LIN {X 0,Y 181.229,Z 745.397,A -85,B 0,C 180,E1 -24524.153,E2 -24524.153} C_VEL
LIN {X 0,Y 171.019,Z 751.513,A -85,B 0,C 180,E1 -24527.303,E2 -24527.303} C_VEL
LIN {X 0,Y 164.032,Z 755.06,A -85,B 0,C 180,E1 -24530.003,E2 -24530.003} C_VEL
LIN {X 0,Y 155.67,Z 758.49,A -85,B 0,C 180,E1 -24534.057,E2 -24534.057} C_VEL
LIN {X 0,Y 149.094,Z 760.427,A -85,B 0,C 180,E1 -24538.049,E2 -24538.049} C_VEL
LIN {X 0,Y 142.632,Z 761.412,A -85,B 0,C 180,E1 -24543.67,E2 -24543.67} C_VEL
LIN {X 0,Y 138.275,Z 760.942,A -85,B 0,C 180,E1 -24549.154,E2 -24549.154} C_VEL
LIN {X 0,Y 135.73,Z 759.131,A -85,B 0,C 180,E1 -24554.99,E2 -24554.99} C_VEL
LIN {X 0,Y 134.847,Z 755.97,A -85,B 0,C 180,E1 -24561,E2 -24561} C_VEL
LIN {X 0,Y 135.175,Z 752.553,A -85,B 0,C 180,E1 -24565.522,E2 -24565.522} C_VEL
LIN {X 0,Y 135.672,Z 749.703,A -85,B 0,C 180,E1 -24568.511,E2 -24568.511} C_VEL
LIN {X 0,Y 135.626,Z 745.103,A -85,B 0,C 180,E1 -24572.222,E2 -24572.222} C_VEL
LIN {X 0,Y 135.586,Z 739.321,A -85,B 0,C 180,E1 -24575.945,E2 -24575.945} C_VEL
LIN {X 0,Y 135.696,Z 732.068,A -85,B 0,C 180,E1 -24579.732,E2 -24579.732} C_VEL
LIN {X 0,Y 136.328,Z 723.561,A -85,B 0,C 180,E1 -24583.409,E2 -24583.409} C_VEL
LIN {X 0,Y 136.604,Z 720.647,A -85,B 0,C 180,E1 -24584.52,E2 -24584.52} C_VEL
LIN {X 0,Y 137.564,Z 713.674,A -85,B 0,C 180,E1 -24589.39,E2 -24589.39} C_VEL
LIN {X 0,Y 139.573,Z 705.628,A -85,B 0,C 180,E1 -24593.75,E2 -24593.75} C_VEL
LIN {X 0,Y 141.934,Z 697.426,A -85,B 0,C 180,E1 -24597.254,E2 -24597.254} C_VEL
LIN {X 0,Y 144.902,Z 687.449,A -85,B 0,C 180,E1 -24600.609,E2 -24600.609} C_VEL
LIN {X 0,Y 148.196,Z 676.409,A -85,B 0,C 180,E1 -24603.451,E2 -24603.451} C_VEL
LIN {X 0,Y 150.997,Z 665.577,A -85,B 0,C 180,E1 -24605.571,E2 -24605.571} C_VEL
LIN {X 0,Y 153.57,Z 653.675,A -85,B 0,C 180,E1 -24607.322,E2 -24607.322} C_VEL
LIN {X 0,Y 155.586,Z 640.822,A -85,B 0,C 180,E1 -24608.701,E2 -24608.701} C_VEL
LIN {X 0,Y 156.825,Z 627.95,A -85,B 0,C 180,E1 -24609.612,E2 -24609.612} C_VEL
LIN {X 0,Y 157.546,Z 613.92,A -85,B 0,C 180,E1 -24610.242,E2 -24610.242} C_VEL
LIN {X 0,Y 155.056,Z 553.997,A -85,B 0,C 180,E1 -24614.23,E2 -24614.23} C_VEL
LIN {X 0,Y 151.174,Z 543.008,A -85,B 0,C 180,E1 -24616.002,E2 -24616.002} C_VEL
LIN {X 0,Y 146.403,Z 531.751,A -85,B 0,C 180,E1 -24618.235,E2 -24618.235} C_VEL
LIN {X 0,Y 142.973,Z 524.786,A -85,B 0,C 180,E1 -24619.906,E2 -24619.906} C_VEL
LIN {X 0,Y 140.588,Z 520.199,A -85,B 0,C 180,E1 -24621.118,E2 -24621.118} C_VEL
LIN {X 0,Y 138.476,Z 515.7,A -85,B 0,C 180,E1 -24622.479,E2 -24622.479} C_VEL
LIN {X 0,Y 136.204,Z 508.223,A -85,B 0,C 180,E1 -24628.068,E2 -24628.068} C_VEL
LIN {X 0,Y 136.07,Z 507.555,A -85,B 0,C 180,E1 -24628.901,E2 -24628.901} C_VEL
LIN {X 0,Y 136.136,Z 507.493,A -85,B 0,C 180,E1 -24632.313,E2 -24632.313} C_VEL
LIN {X 0,Y 136.233,Z 507.491,A -85,B 0,C 180,E1 -24638.83,E2 -24638.83} C_VEL
LIN {X 0,Y 136.273,Z 507.509,A -85,B 0,C 180,E1 -24645.055,E2 -24645.055} C_VEL
LIN {X 0,Y 136.486,Z 507.45,A -85,B 0,C 180,E1 -24648.113,E2 -24648.113} C_VEL
LIN {X 0,Y 136.58,Z 507.448,A -85,B 0,C 180,E1 -24651.119,E2 -24651.119} C_VEL
LIN {X 0,Y 137.122,Z 507.368,A -85,B 0,C 180,E1 -24659.999,E2 -24659.999} C_VEL
LIN {X 0,Y 136.566,Z 507.432,A -85,B 0,C 180,E1 -24668.88,E2 -24668.88} C_VEL
LIN {X 0,Y 136.479,Z 507.466,A -85,B 0,C 180,E1 -24671.954,E2 -24671.954} C_VEL
LIN {X 0,Y 136.239,Z 507.479,A -85,B 0,C 180,E1 -24678.029,E2 -24678.029} C_VEL
LIN {X 0,Y 136.186,Z 507.496,A -85,B 0,C 180,E1 -24681.75,E2 -24681.75} C_VEL
LIN {X 0,Y 136.088,Z 507.498,A -85,B 0,C 180,E1 -24688.618,E2 -24688.618} C_VEL
LIN {X 0,Y 136.059,Z 507.528,A -85,B 0,C 180,E1 -24694.623,E2 -24694.623} C_VEL
LIN {X 0,Y 136.025,Z 507.521,A -85,B 0,C 180,E1 -24699.203,E2 -24699.203} C_VEL
LIN {X 0,Y 136.035,Z 507.52,A -85,B 0,C 180,E1 -24703.681,E2 -24703.681} C_VEL
LIN {X 0,Y 136.08,Z 507.535,A -85,B 0,C 180,E1 -24707.832,E2 -24707.832} C_VEL
LIN {X 0,Y 136.125,Z 507.717,A -85,B 0,C 180,E1 -24711.986,E2 -24711.986} C_VEL
LIN {X 0,Y 136.369,Z 508.823,A -85,B 0,C 180,E1 -24712.654,E2 -24712.654} C_VEL
LIN {X 0,Y 137.916,Z 511.442,A -85,B 0,C 180,E1 -24713.555,E2 -24713.555} C_VEL
LIN {X 0,Y 139.347,Z 513.019,A -85,B 0,C 180,E1 -24714.26,E2 -24714.26} C_VEL
LIN {X 0,Y 141.795,Z 516.64,A -85,B 0,C 180,E1 -24715.486,E2 -24715.486} C_VEL
LIN {X 0,Y 147.533,Z 525.722,A -85,B 0,C 180,E1 -24718.149,E2 -24718.149} C_VEL
LIN {X 0,Y 153.564,Z 536.504,A -85,B 0,C 180,E1 -24720.727,E2 -24720.727} C_VEL
LIN {X 0,Y 159.744,Z 549.453,A -85,B 0,C 180,E1 -24723.189,E2 -24723.189} C_VEL
LIN {X 0,Y 160.42,Z 551.193,A -85,B 0,C 180,E1 -24723.46,E2 -24723.46} C_VEL
LIN {X 0,Y 158.812,Z 593.508,A -85,B 0,C 180,E1 -24725.453,E2 -24725.453} C_VEL
LIN {X 0,Y 157.758,Z 606.514,A -85,B 0,C 180,E1 -24726.542,E2 -24726.542} C_VEL
LIN {X 0,Y 156.131,Z 618.853,A -85,B 0,C 180,E1 -24728.032,E2 -24728.032} C_VEL
LIN {X 0,Y 153.973,Z 630.728,A -85,B 0,C 180,E1 -24729.986,E2 -24729.986} C_VEL
LIN {X 0,Y 151.336,Z 642.124,A -85,B 0,C 180,E1 -24732.436,E2 -24732.436} C_VEL
LIN {X 0,Y 148.657,Z 652.397,A -85,B 0,C 180,E1 -24735.284,E2 -24735.284} C_VEL
LIN {X 0,Y 146.153,Z 660.84,A -85,B 0,C 180,E1 -24738.212,E2 -24738.212} C_VEL
LIN {X 0,Y 143.314,Z 669.988,A -85,B 0,C 180,E1 -24742.254,E2 -24742.254} C_VEL
LIN {X 0,Y 140.794,Z 677.789,A -85,B 0,C 180,E1 -24746.676,E2 -24746.676} C_VEL
LIN {X 0,Y 138.812,Z 684.232,A -85,B 0,C 180,E1 -24751.455,E2 -24751.455} C_VEL
LIN {X 0,Y 137.647,Z 688.768,A -85,B 0,C 180,E1 -24755.866,E2 -24755.866} C_VEL
LIN {X 0,Y 137.075,Z 692.237,A -85,B 0,C 180,E1 -24760.343,E2 -24760.343} C_VEL
LIN {X 0,Y 137.153,Z 694.712,A -85,B 0,C 180,E1 -24764.85,E2 -24764.85} C_VEL
LIN {X 0,Y 138.239,Z 696.548,A -85,B 0,C 180,E1 -24770.852,E2 -24770.852} C_VEL
LIN {X 0,Y 139.867,Z 696.842,A -85,B 0,C 180,E1 -24775.252,E2 -24775.252} C_VEL
LIN {X 0,Y 142.219,Z 696.204,A -85,B 0,C 180,E1 -24779.62,E2 -24779.62} C_VEL
LIN {X 0,Y 144.114,Z 695.281,A -85,B 0,C 180,E1 -24782.447,E2 -24782.447} C_VEL
LIN {X 0,Y 146.406,Z 693.825,A -85,B 0,C 180,E1 -24785.31,E2 -24785.31} C_VEL
LIN {X 0,Y 150.148,Z 690.962,A -85,B 0,C 180,E1 -24789.196,E2 -24789.196} C_VEL
LIN {X 0,Y 155.29,Z 686.157,A -85,B 0,C 180,E1 -24793.606,E2 -24793.606} C_VEL
LIN {X 0,Y 157.794,Z 683.53,A -85,B 0,C 180,E1 -24795.454,E2 -24795.454} C_VEL
LIN {X 0,Y 149.569,Z 684.211,A -85,B 0,C 180,E1 -24798.866,E2 -24798.866} C_VEL
LIN {X 0,Y 140.091,Z 684.215,A -85,B 0,C 180,E1 -24804.767,E2 -24804.767} C_VEL
LIN {X 0,Y 139.135,Z 684.128,A -85,B 0,C 180,E1 -24805.92,E2 -24805.92} C_VEL
LIN {X 0,Y 138.913,Z 685.158,A -85,B 0,C 180,E1 -24806.512,E2 -24806.512} C_VEL
LIN {X 0,Y 137.09,Z 699.044,A -85,B 0,C 180,E1 -24810.341,E2 -24810.341} C_VEL
LIN {X 0,Y 135.806,Z 709.281,A -85,B 0,C 180,E1 -24813.905,E2 -24813.905} C_VEL
LIN {X 0,Y 134.865,Z 718.382,A -85,B 0,C 180,E1 -24817.803,E2 -24817.803} C_VEL
LIN {X 0,Y 134.137,Z 727.119,A -85,B 0,C 180,E1 -24822.467,E2 -24822.467} C_VEL
LIN {X 0,Y 133.895,Z 734.113,A -85,B 0,C 180,E1 -24827.111,E2 -24827.111} C_VEL
LIN {X 0,Y 134.285,Z 740.681,A -85,B 0,C 180,E1 -24832.608,E2 -24832.608} C_VEL
LIN {X 0,Y 135.926,Z 745.974,A -85,B 0,C 180,E1 -24838.52,E2 -24838.52} C_VEL
LIN {X 0,Y 138.001,Z 748.97,A -85,B 0,C 180,E1 -24842.92,E2 -24842.92} C_VEL
LIN {X 0,Y 142.183,Z 751.621,A -85,B 0,C 180,E1 -24848.529,E2 -24848.529} C_VEL
LIN {X 0,Y 147.77,Z 752.801,A -85,B 0,C 180,E1 -24853.758,E2 -24853.758} C_VEL
LIN {X 0,Y 154.776,Z 752.488,A -85,B 0,C 180,E1 -24858.534,E2 -24858.534} C_VEL
LIN {X 0,Y 162.866,Z 750.724,A -85,B 0,C 180,E1 -24862.854,E2 -24862.854} C_VEL
LIN {X 0,Y 172.025,Z 747.379,A -85,B 0,C 180,E1 -24866.706,E2 -24866.706} C_VEL
LIN {X 0,Y 179.516,Z 743.741,A -85,B 0,C 180,E1 -24869.3,E2 -24869.3} C_VEL
LIN {X 0,Y 187.457,Z 739.108,A -85,B 0,C 180,E1 -24871.661,E2 -24871.661} C_VEL
LIN {X 0,Y 196.841,Z 732.461,A -85,B 0,C 180,E1 -24874.06,E2 -24874.06} C_VEL
LIN {X 0,Y 205.986,Z 724.791,A -85,B 0,C 180,E1 -24876.055,E2 -24876.055} C_VEL
LIN {X 0,Y 211.642,Z 719.272,A -85,B 0,C 180,E1 -24877.154,E2 -24877.154} C_VEL
LIN {X 0,Y 212.865,Z 718.031,A -85,B 0,C 180,E1 -24877.586,E2 -24877.586} C_VEL
LIN {X 0,Y 203.705,Z 727.465,A -85,B 0,C 180,E1 -24879.075,E2 -24879.075} C_VEL
LIN {X 0,Y 199.807,Z 731.054,A -85,B 0,C 180,E1 -24879.811,E2 -24879.811} C_VEL
LIN {X 0,Y 195.562,Z 734.617,A -85,B 0,C 180,E1 -24880.454,E2 -24880.454} C_VEL
LIN {X 0,Y 187.687,Z 740.276,A -85,B 0,C 180,E1 -24881.137,E2 -24881.137} C_VEL
LIN {X 0,Y 179.639,Z 745.219,A -85,B 0,C 180,E1 -24881.969,E2 -24881.969} C_VEL
LIN {X 0,Y 175.187,Z 747.737,A -85,B 0,C 180,E1 -24882.866,E2 -24882.866} C_VEL
LIN {X 0,Y 165.932,Z 752.571,A -85,B 0,C 180,E1 -24885.66,E2 -24885.66} C_VEL
LIN {X 0,Y 158.69,Z 755.703,A -85,B 0,C 180,E1 -24888.365,E2 -24888.365} C_VEL
LIN {X 0,Y 149.985,Z 758.707,A -85,B 0,C 180,E1 -24892.466,E2 -24892.466} C_VEL
LIN {X 0,Y 142.55,Z 760.354,A -85,B 0,C 180,E1 -24896.946,E2 -24896.946} C_VEL
LIN {X 0,Y 136.305,Z 760.804,A -85,B 0,C 180,E1 -24902.346,E2 -24902.346} C_VEL
LIN {X 0,Y 131.704,Z 759.946,A -85,B 0,C 180,E1 -24908.061,E2 -24908.061} C_VEL
LIN {X 0,Y 128.973,Z 757.854,A -85,B 0,C 180,E1 -24914.184,E2 -24914.184} C_VEL
LIN {X 0,Y 128.004,Z 754.352,A -85,B 0,C 180,E1 -24920.514,E2 -24920.514} C_VEL
LIN {X 0,Y 128.351,Z 750.743,A -85,B 0,C 180,E1 -24925.284,E2 -24925.284} C_VEL
LIN {X 0,Y 128.845,Z 747.668,A -85,B 0,C 180,E1 -24928.432,E2 -24928.432} C_VEL
LIN {X 0,Y 128.784,Z 741.622,A -85,B 0,C 180,E1 -24933.123,E2 -24933.123} C_VEL
LIN {X 0,Y 128.752,Z 733.802,A -85,B 0,C 180,E1 -24937.838,E2 -24937.838} C_VEL
LIN {X 0,Y 129.123,Z 725.691,A -85,B 0,C 180,E1 -24941.783,E2 -24941.783} C_VEL
LIN {X 0,Y 129.477,Z 721.14,A -85,B 0,C 180,E1 -24943.732,E2 -24943.732} C_VEL
LIN {X 0,Y 130.27,Z 714.515,A -85,B 0,C 180,E1 -24948.881,E2 -24948.881} C_VEL
LIN {X 0,Y 132.17,Z 706.9,A -85,B 0,C 180,E1 -24953.498,E2 -24953.498} C_VEL
LIN {X 0,Y 134.642,Z 698.606,A -85,B 0,C 180,E1 -24957.454,E2 -24957.454} C_VEL
LIN {X 0,Y 137.731,Z 688.798,A -85,B 0,C 180,E1 -24961.102,E2 -24961.102} C_VEL
LIN {X 0,Y 141.14,Z 678.275,A -85,B 0,C 180,E1 -24964.063,E2 -24964.063} C_VEL
LIN {X 0,Y 144.364,Z 666.543,A -85,B 0,C 180,E1 -24966.604,E2 -24966.604} C_VEL
LIN {X 0,Y 147.032,Z 655.291,A -85,B 0,C 180,E1 -24968.411,E2 -24968.411} C_VEL
LIN {X 0,Y 149.255,Z 642.587,A -85,B 0,C 180,E1 -24969.902,E2 -24969.902} C_VEL
LIN {X 0,Y 150.774,Z 628.997,A -85,B 0,C 180,E1 -24970.988,E2 -24970.988} C_VEL
LIN {X 0,Y 151.631,Z 614.609,A -85,B 0,C 180,E1 -24971.675,E2 -24971.675} C_VEL
LIN {X 0,Y 149.494,Z 556.216,A -85,B 0,C 180,E1 -24975.709,E2 -24975.709} C_VEL
LIN {X 0,Y 145.779,Z 545.595,A -85,B 0,C 180,E1 -24977.549,E2 -24977.549} C_VEL
LIN {X 0,Y 140.792,Z 533.824,A -85,B 0,C 180,E1 -24980.095,E2 -24980.095} C_VEL
LIN {X 0,Y 136.234,Z 524.565,A -85,B 0,C 180,E1 -24982.57,E2 -24982.57} C_VEL
LIN {X 0,Y 133.372,Z 519.261,A -85,B 0,C 180,E1 -24984.224,E2 -24984.224} C_VEL
LIN {X 0,Y 130.784,Z 514.341,A -85,B 0,C 180,E1 -24985.998,E2 -24985.998} C_VEL
LIN {X 0,Y 129.054,Z 508.495,A -85,B 0,C 180,E1 -24990.93,E2 -24990.93} C_VEL
LIN {X 0,Y 129.02,Z 508.389,A -85,B 0,C 180,E1 -24994.164,E2 -24994.164} C_VEL
LIN {X 0,Y 129.097,Z 508.389,A -85,B 0,C 180,E1 -24997.725,E2 -24997.725} C_VEL
LIN {X 0,Y 129.149,Z 508.368,A -85,B 0,C 180,E1 -25000.942,E2 -25000.942} C_VEL
LIN {X 0,Y 129.405,Z 508.332,A -85,B 0,C 180,E1 -25007.818,E2 -25007.818} C_VEL
LIN {X 0,Y 129.505,Z 508.323,A -85,B 0,C 180,E1 -25010.629,E2 -25010.629} C_VEL
LIN {X 0,Y 130.077,Z 508.244,A -85,B 0,C 180,E1 -25019.999,E2 -25019.999} C_VEL
LIN {X 0,Y 129.495,Z 508.311,A -85,B 0,C 180,E1 -25029.369,E2 -25029.369} C_VEL
LIN {X 0,Y 129.381,Z 508.356,A -85,B 0,C 180,E1 -25032.548,E2 -25032.548} C_VEL
LIN {X 0,Y 129.147,Z 508.357,A -85,B 0,C 180,E1 -25039.056,E2 -25039.056} C_VEL
LIN {X 0,Y 129.096,Z 508.386,A -85,B 0,C 180,E1 -25042.399,E2 -25042.399} C_VEL
LIN {X 0,Y 129.018,Z 508.4,A -85,B 0,C 180,E1 -25045.834,E2 -25045.834} C_VEL
LIN {X 0,Y 129.004,Z 508.38,A -85,B 0,C 180,E1 -25049.36,E2 -25049.36} C_VEL
LIN {X 0,Y 128.969,Z 508.402,A -85,B 0,C 180,E1 -25055.184,E2 -25055.184} C_VEL
LIN {X 0,Y 128.97,Z 508.419,A -85,B 0,C 180,E1 -25060.836,E2 -25060.836} C_VEL
LIN {X 0,Y 129.011,Z 508.405,A -85,B 0,C 180,E1 -25067.09,E2 -25067.09} C_VEL
LIN {X 0,Y 129.064,Z 508.734,A -85,B 0,C 180,E1 -25068.766,E2 -25068.766} C_VEL
LIN {X 0,Y 129.373,Z 509.954,A -85,B 0,C 180,E1 -25069.421,E2 -25069.421} C_VEL
LIN {X 0,Y 131.114,Z 512.578,A -85,B 0,C 180,E1 -25070.551,E2 -25070.551} C_VEL
LIN {X 0,Y 132.475,Z 514.021,A -85,B 0,C 180,E1 -25071.327,E2 -25071.327} C_VEL
LIN {X 0,Y 134.708,Z 517.373,A -85,B 0,C 180,E1 -25072.622,E2 -25072.622} C_VEL
LIN {X 0,Y 136.153,Z 519.485,A -85,B 0,C 180,E1 -25073.412,E2 -25073.412} C_VEL
LIN {X 0,Y 141.454,Z 527.468,A -85,B 0,C 180,E1 -25076.104,E2 -25076.104} C_VEL
LIN {X 0,Y 148.043,Z 539.079,A -85,B 0,C 180,E1 -25079.168,E2 -25079.168} C_VEL
LIN {X 0,Y 154.555,Z 552.964,A -85,B 0,C 180,E1 -25081.98,E2 -25081.98} C_VEL
LIN {X 0,Y 152.942,Z 594.325,A -85,B 0,C 180,E1 -25084.01,E2 -25084.01} C_VEL
LIN {X 0,Y 151.835,Z 607.269,A -85,B 0,C 180,E1 -25085.122,E2 -25085.122} C_VEL
LIN {X 0,Y 150.051,Z 620.144,A -85,B 0,C 180,E1 -25086.727,E2 -25086.727} C_VEL
LIN {X 0,Y 147.77,Z 631.93,A -85,B 0,C 180,E1 -25088.742,E2 -25088.742} C_VEL
LIN {X 0,Y 144.996,Z 643.285,A -85,B 0,C 180,E1 -25091.275,E2 -25091.275} C_VEL
LIN {X 0,Y 142.163,Z 653.53,A -85,B 0,C 180,E1 -25094.228,E2 -25094.228} C_VEL
LIN {X 0,Y 139.26,Z 662.771,A -85,B 0,C 180,E1 -25097.62,E2 -25097.62} C_VEL
LIN {X 0,Y 136.318,Z 671.744,A -85,B 0,C 180,E1 -25101.854,E2 -25101.854} C_VEL
LIN {X 0,Y 133.809,Z 679.105,A -85,B 0,C 180,E1 -25106.295,E2 -25106.295} C_VEL
LIN {X 0,Y 132.201,Z 683.961,A -85,B 0,C 180,E1 -25110.005,E2 -25110.005} C_VEL
LIN {X 0,Y 130.85,Z 688.777,A -85,B 0,C 180,E1 -25114.626,E2 -25114.626} C_VEL
LIN {X 0,Y 130.116,Z 692.495,A -85,B 0,C 180,E1 -25119.33,E2 -25119.33} C_VEL
LIN {X 0,Y 130.036,Z 694.856,A -85,B 0,C 180,E1 -25123.389,E2 -25123.389} C_VEL
LIN {X 0,Y 130.668,Z 696.952,A -85,B 0,C 180,E1 -25128.832,E2 -25128.832} C_VEL
LIN {X 0,Y 131.492,Z 697.628,A -85,B 0,C 180,E1 -25131.976,E2 -25131.976} C_VEL
LIN {X 0,Y 133.16,Z 697.836,A -85,B 0,C 180,E1 -25136.206,E2 -25136.206} C_VEL
LIN {X 0,Y 135.932,Z 697.104,A -85,B 0,C 180,E1 -25141.138,E2 -25141.138} C_VEL
LIN {X 0,Y 138.017,Z 696.11,A -85,B 0,C 180,E1 -25144.071,E2 -25144.071} C_VEL
LIN {X 0,Y 140.431,Z 694.643,A -85,B 0,C 180,E1 -25146.915,E2 -25146.915} C_VEL
LIN {X 0,Y 144.56,Z 691.615,A -85,B 0,C 180,E1 -25151.026,E2 -25151.026} C_VEL
LIN {X 0,Y 149.604,Z 687.132,A -85,B 0,C 180,E1 -25155.199,E2 -25155.199} C_VEL
LIN {X 0,Y 144.92,Z 687.539,A -85,B 0,C 180,E1 -25157.241,E2 -25157.241} C_VEL
LIN {X 0,Y 136.909,Z 687.782,A -85,B 0,C 180,E1 -25161.977,E2 -25161.977} C_VEL
LIN {X 0,Y 131.712,Z 687.513,A -85,B 0,C 180,E1 -25166.387,E2 -25166.387} C_VEL
LIN {X 0,Y 131.451,Z 687.871,A -85,B 0,C 180,E1 -25167.113,E2 -25167.113} C_VEL
LIN {X 0,Y 131.075,Z 690.333,A -85,B 0,C 180,E1 -25167.932,E2 -25167.932} C_VEL
LIN {X 0,Y 129.543,Z 702.181,A -85,B 0,C 180,E1 -25171.661,E2 -25171.661} C_VEL
LIN {X 0,Y 128.315,Z 712.571,A -85,B 0,C 180,E1 -25175.747,E2 -25175.747} C_VEL
LIN {X 0,Y 127.444,Z 721.617,A -85,B 0,C 180,E1 -25180.152,E2 -25180.152} C_VEL
LIN {X 0,Y 126.996,Z 729.346,A -85,B 0,C 180,E1 -25184.761,E2 -25184.761} C_VEL
LIN {X 0,Y 126.92,Z 734.88,A -85,B 0,C 180,E1 -25188.826,E2 -25188.826} C_VEL
LIN {X 0,Y 127.469,Z 740.353,A -85,B 0,C 180,E1 -25193.67,E2 -25193.67} C_VEL
LIN {X 0,Y 128.753,Z 744.741,A -85,B 0,C 180,E1 -25198.437,E2 -25198.437} C_VEL
LIN {X 0,Y 130.814,Z 748.13,A -85,B 0,C 180,E1 -25203.081,E2 -25203.081} C_VEL
LIN {X 0,Y 135.324,Z 751.497,A -85,B 0,C 180,E1 -25209.307,E2 -25209.307} C_VEL
LIN {X 0,Y 140.756,Z 753.082,A -85,B 0,C 180,E1 -25214.458,E2 -25214.458} C_VEL
LIN {X 0,Y 147.945,Z 753.363,A -85,B 0,C 180,E1 -25219.423,E2 -25219.423} C_VEL
LIN {X 0,Y 156.26,Z 752.231,A -85,B 0,C 180,E1 -25223.879,E2 -25223.879} C_VEL
LIN {X 0,Y 165.706,Z 749.512,A -85,B 0,C 180,E1 -25227.811,E2 -25227.811} C_VEL
LIN {X 0,Y 173.368,Z 746.484,A -85,B 0,C 180,E1 -25230.447,E2 -25230.447} C_VEL
LIN {X 0,Y 181.509,Z 742.423,A -85,B 0,C 180,E1 -25232.826,E2 -25232.826} C_VEL
LIN {X 0,Y 190.977,Z 736.694,A -85,B 0,C 180,E1 -25235.189,E2 -25235.189} C_VEL
LIN {X 0,Y 199.017,Z 730.882,A -85,B 0,C 180,E1 -25236.895,E2 -25236.895} C_VEL
LIN {X 0,Y 199.44,Z 730.626,A -85,B 0,C 180,E1 -25237.541,E2 -25237.541} C_VEL
LIN {X 0,Y 189.089,Z 738.801,A -85,B 0,C 180,E1 -25239.531,E2 -25239.531} C_VEL
LIN {X 0,Y 179.189,Z 745.392,A -85,B 0,C 180,E1 -25241.819,E2 -25241.819} C_VEL
LIN {X 0,Y 175.187,Z 747.737,A -85,B 0,C 180,E1 -25242.866,E2 -25242.866} C_VEL
LIN {X 0,Y 170.662,Z 750.117,A -85,B 0,C 180,E1 -25243.871,E2 -25243.871} C_VEL
LIN {X 0,Y 162.216,Z 753.567,A -85,B 0,C 180,E1 -25245.23,E2 -25245.23} C_VEL
LIN {X 0,Y 153.855,Z 756.24,A -85,B 0,C 180,E1 -25246.84,E2 -25246.84} C_VEL
LIN {X 0,Y 149.549,Z 757.423,A -85,B 0,C 180,E1 -25248.257,E2 -25248.257} C_VEL
LIN {X 0,Y 140.228,Z 759.572,A -85,B 0,C 180,E1 -25253.023,E2 -25253.023} C_VEL
LIN {X 0,Y 133.109,Z 760.234,A -85,B 0,C 180,E1 -25258.125,E2 -25258.125} C_VEL
LIN {X 0,Y 127.483,Z 759.652,A -85,B 0,C 180,E1 -25263.825,E2 -25263.825} C_VEL
LIN {X 0,Y 123.531,Z 757.802,A -85,B 0,C 180,E1 -25270.035,E2 -25270.035} C_VEL
LIN {X 0,Y 121.49,Z 754.698,A -85,B 0,C 180,E1 -25276.615,E2 -25276.615} C_VEL
LIN {X 0,Y 121.362,Z 750.131,A -85,B 0,C 180,E1 -25283.344,E2 -25283.344} C_VEL
LIN {X 0,Y 122.042,Z 745.526,A -85,B 0,C 180,E1 -25288.345,E2 -25288.345} C_VEL
LIN {X 0,Y 121.949,Z 740.256,A -85,B 0,C 180,E1 -25292.472,E2 -25292.472} C_VEL
LIN {X 0,Y 121.881,Z 733.713,A -85,B 0,C 180,E1 -25296.617,E2 -25296.617} C_VEL
LIN {X 0,Y 122.225,Z 724.042,A -85,B 0,C 180,E1 -25301.572,E2 -25301.572} C_VEL
LIN {X 0,Y 122.352,Z 721.696,A -85,B 0,C 180,E1 -25302.658,E2 -25302.658} C_VEL
LIN {X 0,Y 123.016,Z 715.262,A -85,B 0,C 180,E1 -25308.308,E2 -25308.308} C_VEL
LIN {X 0,Y 124.753,Z 708.085,A -85,B 0,C 180,E1 -25313.219,E2 -25313.219} C_VEL
LIN {X 0,Y 127.58,Z 699.051,A -85,B 0,C 180,E1 -25317.959,E2 -25317.959} C_VEL
LIN {X 0,Y 130.947,Z 688.99,A -85,B 0,C 180,E1 -25321.999,E2 -25321.999} C_VEL
LIN {X 0,Y 134.448,Z 678.77,A -85,B 0,C 180,E1 -25325.093,E2 -25325.093} C_VEL
LIN {X 0,Y 137.798,Z 667.365,A -85,B 0,C 180,E1 -25327.729,E2 -25327.729} C_VEL
LIN {X 0,Y 140.772,Z 655.577,A -85,B 0,C 180,E1 -25329.76,E2 -25329.76} C_VEL
LIN {X 0,Y 143.235,Z 642.744,A -85,B 0,C 180,E1 -25331.358,E2 -25331.358} C_VEL
LIN {X 0,Y 144.873,Z 629.088,A -85,B 0,C 180,E1 -25332.517,E2 -25332.517} C_VEL
LIN {X 0,Y 145.807,Z 615.613,A -85,B 0,C 180,E1 -25333.193,E2 -25333.193} C_VEL
LIN {X 0,Y 144.01,Z 558.309,A -85,B 0,C 180,E1 -25337.319,E2 -25337.319} C_VEL
LIN {X 0,Y 139.806,Z 546.37,A -85,B 0,C 180,E1 -25339.594,E2 -25339.594} C_VEL
LIN {X 0,Y 134.923,Z 535.031,A -85,B 0,C 180,E1 -25342.349,E2 -25342.349} C_VEL
LIN {X 0,Y 129.935,Z 524.856,A -85,B 0,C 180,E1 -25345.405,E2 -25345.405} C_VEL
LIN {X 0,Y 126.142,Z 518.268,A -85,B 0,C 180,E1 -25347.923,E2 -25347.923} C_VEL
LIN {X 0,Y 123.07,Z 512.77,A -85,B 0,C 180,E1 -25350.375,E2 -25350.375} C_VEL
LIN {X 0,Y 122.019,Z 509.465,A -85,B 0,C 180,E1 -25353.487,E2 -25353.487} C_VEL
LIN {X 0,Y 122.038,Z 509.252,A -85,B 0,C 180,E1 -25359.784,E2 -25359.784} C_VEL
LIN {X 0,Y 122.253,Z 509.23,A -85,B 0,C 180,E1 -25366.705,E2 -25366.705} C_VEL
LIN {X 0,Y 122.435,Z 509.198,A -85,B 0,C 180,E1 -25370.083,E2 -25370.083} C_VEL
LIN {X 0,Y 122.592,Z 509.18,A -85,B 0,C 180,E1 -25376.712,E2 -25376.712} C_VEL
LIN {X 0,Y 123.031,Z 509.12,A -85,B 0,C 180,E1 -25379.999,E2 -25379.999} C_VEL
LIN {X 0,Y 122.399,Z 509.201,A -85,B 0,C 180,E1 -25387.145,E2 -25387.145} C_VEL
LIN {X 0,Y 122.35,Z 509.228,A -85,B 0,C 180,E1 -25392.471,E2 -25392.471} C_VEL
LIN {X 0,Y 122.105,Z 509.248,A -85,B 0,C 180,E1 -25396.724,E2 -25396.724} C_VEL
LIN {X 0,Y 122.016,Z 509.272,A -85,B 0,C 180,E1 -25402.857,E2 -25402.857} C_VEL
LIN {X 0,Y 121.93,Z 509.264,A -85,B 0,C 180,E1 -25407.458,E2 -25407.458} C_VEL
LIN {X 0,Y 121.895,Z 509.277,A -85,B 0,C 180,E1 -25411.258,E2 -25411.258} C_VEL
LIN {X 0,Y 121.887,Z 509.275,A -85,B 0,C 180,E1 -25416.183,E2 -25416.183} C_VEL
LIN {X 0,Y 121.902,Z 509.301,A -85,B 0,C 180,E1 -25421.463,E2 -25421.463} C_VEL
LIN {X 0,Y 121.945,Z 509.557,A -85,B 0,C 180,E1 -25424.645,E2 -25424.645} C_VEL
LIN {X 0,Y 122.237,Z 510.661,A -85,B 0,C 180,E1 -25425.409,E2 -25425.409} C_VEL
LIN {X 0,Y 123.774,Z 513.201,A -85,B 0,C 180,E1 -25426.633,E2 -25426.633} C_VEL
LIN {X 0,Y 125.622,Z 514.905,A -85,B 0,C 180,E1 -25427.868,E2 -25427.868} C_VEL
LIN {X 0,Y 127.726,Z 518.179,A -85,B 0,C 180,E1 -25429.313,E2 -25429.313} C_VEL
LIN {X 0,Y 129.124,Z 519.906,A -85,B 0,C 180,E1 -25430.181,E2 -25430.181} C_VEL
LIN {X 0,Y 134.391,Z 527.686,A -85,B 0,C 180,E1 -25433.269,E2 -25433.269} C_VEL
LIN {X 0,Y 139.727,Z 536.513,A -85,B 0,C 180,E1 -25436.079,E2 -25436.079} C_VEL
LIN {X 0,Y 144.984,Z 546.623,A -85,B 0,C 180,E1 -25438.634,E2 -25438.634} C_VEL
LIN {X 0,Y 148.918,Z 555.258,A -85,B 0,C 180,E1 -25440.452,E2 -25440.452} C_VEL
LIN {X 0,Y 147.152,Z 595.408,A -85,B 0,C 180,E1 -25442.472,E2 -25442.472} C_VEL
LIN {X 0,Y 145.981,Z 608.403,A -85,B 0,C 180,E1 -25443.632,E2 -25443.632} C_VEL
LIN {X 0,Y 144.229,Z 620.345,A -85,B 0,C 180,E1 -25445.153,E2 -25445.153} C_VEL
LIN {X 0,Y 141.992,Z 631.566,A -85,B 0,C 180,E1 -25447.065,E2 -25447.065} C_VEL
LIN {X 0,Y 139.058,Z 643.171,A -85,B 0,C 180,E1 -25449.673,E2 -25449.673} C_VEL
LIN {X 0,Y 136.047,Z 653.598,A -85,B 0,C 180,E1 -25452.726,E2 -25452.726} C_VEL
LIN {X 0,Y 132.961,Z 663.043,A -85,B 0,C 180,E1 -25456.245,E2 -25456.245} C_VEL
LIN {X 0,Y 129.789,Z 672.144,A -85,B 0,C 180,E1 -25460.656,E2 -25460.656} C_VEL
LIN {X 0,Y 127.306,Z 678.922,A -85,B 0,C 180,E1 -25464.826,E2 -25464.826} C_VEL
LIN {X 0,Y 125.094,Z 685.47,A -85,B 0,C 180,E1 -25470.005,E2 -25470.005} C_VEL
LIN {X 0,Y 123.705,Z 690.184,A -85,B 0,C 180,E1 -25474.894,E2 -25474.894} C_VEL
LIN {X 0,Y 123.041,Z 693.8,A -85,B 0,C 180,E1 -25479.872,E2 -25479.872} C_VEL
LIN {X 0,Y 123.006,Z 695.886,A -85,B 0,C 180,E1 -25483.766,E2 -25483.766} C_VEL
LIN {X 0,Y 123.855,Z 698.076,A -85,B 0,C 180,E1 -25489.911,E2 -25489.911} C_VEL
LIN {X 0,Y 124.8,Z 698.675,A -85,B 0,C 180,E1 -25493.222,E2 -25493.222} C_VEL
LIN {X 0,Y 127.77,Z 698.621,A -85,B 0,C 180,E1 -25499.678,E2 -25499.678} C_VEL
LIN {X 0,Y 129.77,Z 697.996,A -85,B 0,C 180,E1 -25502.797,E2 -25502.797} C_VEL
LIN {X 0,Y 134.093,Z 695.755,A -85,B 0,C 180,E1 -25508.173,E2 -25508.173} C_VEL
LIN {X 0,Y 139.123,Z 692.27,A -85,B 0,C 180,E1 -25513.004,E2 -25513.004} C_VEL
LIN {X 0,Y 140.752,Z 690.983,A -85,B 0,C 180,E1 -25514.356,E2 -25514.356} C_VEL
LIN {X 0,Y 140.256,Z 690.513,A -85,B 0,C 180,E1 -25515.453,E2 -25515.453} C_VEL
LIN {X 0,Y 131.964,Z 690.972,A -85,B 0,C 180,E1 -25520.278,E2 -25520.278} C_VEL
LIN {X 0,Y 124,Z 690.732,A -85,B 0,C 180,E1 -25527.594,E2 -25527.594} C_VEL
LIN {X 0,Y 123.794,Z 691.458,A -85,B 0,C 180,E1 -25528.393,E2 -25528.393} C_VEL
LIN {X 0,Y 122.116,Z 704.804,A -85,B 0,C 180,E1 -25533.051,E2 -25533.051} C_VEL
LIN {X 0,Y 120.926,Z 715.427,A -85,B 0,C 180,E1 -25537.703,E2 -25537.703} C_VEL
LIN {X 0,Y 120.25,Z 723.579,A -85,B 0,C 180,E1 -25542.133,E2 -25542.133} C_VEL
LIN {X 0,Y 119.96,Z 731.262,A -85,B 0,C 180,E1 -25547.31,E2 -25547.31} C_VEL
LIN {X 0,Y 120.35,Z 738.394,A -85,B 0,C 180,E1 -25553.294,E2 -25553.294} C_VEL
LIN {X 0,Y 121.613,Z 743.231,A -85,B 0,C 180,E1 -25558.345,E2 -25558.345} C_VEL
LIN {X 0,Y 124.543,Z 748.152,A -85,B 0,C 180,E1 -25564.857,E2 -25564.857} C_VEL
LIN {X 0,Y 128.568,Z 751.203,A -85,B 0,C 180,E1 -25570.253,E2 -25570.253} C_VEL
LIN {X 0,Y 133.747,Z 753.126,A -85,B 0,C 180,E1 -25575.234,E2 -25575.234} C_VEL
LIN {X 0,Y 141.132,Z 754.006,A -85,B 0,C 180,E1 -25580.402,E2 -25580.402} C_VEL
LIN {X 0,Y 149.677,Z 753.484,A -85,B 0,C 180,E1 -25584.999,E2 -25584.999} C_VEL
LIN {X 0,Y 159.409,Z 751.436,A -85,B 0,C 180,E1 -25589.011,E2 -25589.011} C_VEL
LIN {X 0,Y 167.255,Z 748.929,A -85,B 0,C 180,E1 -25591.686,E2 -25591.686} C_VEL
LIN {X 0,Y 178.797,Z 743.963,A -85,B 0,C 180,E1 -25594.885,E2 -25594.885} C_VEL
LIN {X 0,Y 187.367,Z 739.251,A -85,B 0,C 180,E1 -25596.881,E2 -25596.881} C_VEL
LIN {X 0,Y 186.244,Z 740.052,A -85,B 0,C 180,E1 -25597.58,E2 -25597.58} C_VEL
LIN {X 0,Y 176.718,Z 745.884,A -85,B 0,C 180,E1 -25599.607,E2 -25599.607} C_VEL
LIN {X 0,Y 166.294,Z 751.171,A -85,B 0,C 180,E1 -25602.298,E2 -25602.298} C_VEL
LIN {X 0,Y 158.435,Z 754.477,A -85,B 0,C 180,E1 -25604.781,E2 -25604.781} C_VEL
LIN {X 0,Y 149.549,Z 757.423,A -85,B 0,C 180,E1 -25608.257,E2 -25608.257} C_VEL
LIN {X 0,Y 145.321,Z 758.452,A -85,B 0,C 180,E1 -25609.814,E2 -25609.814} C_VEL
LIN {X 0,Y 137.369,Z 759.459,A -85,B 0,C 180,E1 -25612.181,E2 -25612.181} C_VEL
LIN {X 0,Y 129.861,Z 759.676,A -85,B 0,C 180,E1 -25614.917,E2 -25614.917} C_VEL
LIN {X 0,Y 126.438,Z 759.483,A -85,B 0,C 180,E1 -25617.047,E2 -25617.047} C_VEL
LIN {X 0,Y 121.19,Z 758.61,A -85,B 0,C 180,E1 -25622.353,E2 -25622.353} C_VEL
LIN {X 0,Y 116.988,Z 756.454,A -85,B 0,C 180,E1 -25628.866,E2 -25628.866} C_VEL
LIN {X 0,Y 114.79,Z 752.958,A -85,B 0,C 180,E1 -25635.818,E2 -25635.818} C_VEL
LIN {X 0,Y 114.636,Z 748.069,A -85,B 0,C 180,E1 -25642.951,E2 -25642.951} C_VEL
LIN {X 0,Y 115.112,Z 744.959,A -85,B 0,C 180,E1 -25646.494,E2 -25646.494} C_VEL
LIN {X 0,Y 115.254,Z 742.131,A -85,B 0,C 180,E1 -25649.121,E2 -25649.121} C_VEL
LIN {X 0,Y 115.073,Z 736.306,A -85,B 0,C 180,E1 -25653.496,E2 -25653.496} C_VEL
LIN {X 0,Y 114.991,Z 729.05,A -85,B 0,C 180,E1 -25657.898,E2 -25657.898} C_VEL
LIN {X 0,Y 115.326,Z 722.07,A -85,B 0,C 180,E1 -25661.543,E2 -25661.543} C_VEL
LIN {X 0,Y 115.739,Z 715.909,A -85,B 0,C 180,E1 -25667.669,E2 -25667.669} C_VEL
LIN {X 0,Y 117.376,Z 709.083,A -85,B 0,C 180,E1 -25672.898,E2 -25672.898} C_VEL
LIN {X 0,Y 120.134,Z 700.658,A -85,B 0,C 180,E1 -25677.899,E2 -25677.899} C_VEL
LIN {X 0,Y 123.175,Z 692.07,A -85,B 0,C 180,E1 -25681.849,E2 -25681.849} C_VEL
LIN {X 0,Y 126.957,Z 681.533,A -85,B 0,C 180,E1 -25685.532,E2 -25685.532} C_VEL
LIN {X 0,Y 130.838,Z 669.662,A -85,B 0,C 180,E1 -25688.634,E2 -25688.634} C_VEL
LIN {X 0,Y 134.102,Z 657.803,A -85,B 0,C 180,E1 -25690.92,E2 -25690.92} C_VEL
LIN {X 0,Y 136.691,Z 645.977,A -85,B 0,C 180,E1 -25692.583,E2 -25692.583} C_VEL
LIN {X 0,Y 138.701,Z 632.742,A -85,B 0,C 180,E1 -25693.907,E2 -25693.907} C_VEL
LIN {X 0,Y 139.93,Z 619.903,A -85,B 0,C 180,E1 -25694.673,E2 -25694.673} C_VEL
LIN {X 0,Y 139.963,Z 611.462,A -85,B 0,C 180,E1 -25695.205,E2 -25695.205} C_VEL
LIN {X 0,Y 138.615,Z 560.34,A -85,B 0,C 180,E1 -25699.072,E2 -25699.072} C_VEL
LIN {X 0,Y 134.319,Z 548.06,A -85,B 0,C 180,E1 -25701.629,E2 -25701.629} C_VEL
LIN {X 0,Y 129.756,Z 537.481,A -85,B 0,C 180,E1 -25704.476,E2 -25704.476} C_VEL
LIN {X 0,Y 125.553,Z 528.831,A -85,B 0,C 180,E1 -25707.324,E2 -25707.324} C_VEL
LIN {X 0,Y 122.489,Z 523.211,A -85,B 0,C 180,E1 -25709.576,E2 -25709.576} C_VEL
LIN {X 0,Y 118.998,Z 517.241,A -85,B 0,C 180,E1 -25712.399,E2 -25712.399} C_VEL
LIN {X 0,Y 115.282,Z 511.674,A -85,B 0,C 180,E1 -25715.847,E2 -25715.847} C_VEL
LIN {X 0,Y 115.001,Z 510.433,A -85,B 0,C 180,E1 -25716.885,E2 -25716.885} C_VEL
LIN {X 0,Y 114.971,Z 510.138,A -85,B 0,C 180,E1 -25718.482,E2 -25718.482} C_VEL
LIN {X 0,Y 115.137,Z 510.125,A -85,B 0,C 180,E1 -25725.866,E2 -25725.866} C_VEL
LIN {X 0,Y 115.353,Z 510.077,A -85,B 0,C 180,E1 -25729.467,E2 -25729.467} C_VEL
LIN {X 0,Y 115.518,Z 510.061,A -85,B 0,C 180,E1 -25736.511,E2 -25736.511} C_VEL
LIN {X 0,Y 115.983,Z 509.996,A -85,B 0,C 180,E1 -25739.999,E2 -25739.999} C_VEL
LIN {X 0,Y 115.367,Z 510.076,A -85,B 0,C 180,E1 -25747.035,E2 -25747.035} C_VEL
LIN {X 0,Y 115.271,Z 510.111,A -85,B 0,C 180,E1 -25752.735,E2 -25752.735} C_VEL
LIN {X 0,Y 115.005,Z 510.121,A -85,B 0,C 180,E1 -25757.79,E2 -25757.79} C_VEL
LIN {X 0,Y 114.936,Z 510.162,A -85,B 0,C 180,E1 -25763.495,E2 -25763.495} C_VEL
LIN {X 0,Y 114.85,Z 510.151,A -85,B 0,C 180,E1 -25771.064,E2 -25771.064} C_VEL
LIN {X 0,Y 114.827,Z 510.239,A -85,B 0,C 180,E1 -25778.853,E2 -25778.853} C_VEL
LIN {X 0,Y 115.001,Z 511.064,A -85,B 0,C 180,E1 -25780.201,E2 -25780.201} C_VEL
LIN {X 0,Y 116.564,Z 513.994,A -85,B 0,C 180,E1 -25781.896,E2 -25781.896} C_VEL
LIN {X 0,Y 118.91,Z 515.962,A -85,B 0,C 180,E1 -25783.797,E2 -25783.797} C_VEL
LIN {X 0,Y 120.856,Z 519.153,A -85,B 0,C 180,E1 -25785.421,E2 -25785.421} C_VEL
LIN {X 0,Y 122.572,Z 521.004,A -85,B 0,C 180,E1 -25786.668,E2 -25786.668} C_VEL
LIN {X 0,Y 125.037,Z 524.484,A -85,B 0,C 180,E1 -25788.415,E2 -25788.415} C_VEL
LIN {X 0,Y 130.672,Z 533.023,A -85,B 0,C 180,E1 -25792.006,E2 -25792.006} C_VEL
LIN {X 0,Y 135.568,Z 541.402,A -85,B 0,C 180,E1 -25794.789,E2 -25794.789} C_VEL
LIN {X 0,Y 140.481,Z 551.149,A -85,B 0,C 180,E1 -25797.364,E2 -25797.364} C_VEL
LIN {X 0,Y 143.299,Z 557.454,A -85,B 0,C 180,E1 -25798.767,E2 -25798.767} C_VEL
LIN {X 0,Y 141.432,Z 596.902,A -85,B 0,C 180,E1 -25800.835,E2 -25800.835} C_VEL
LIN {X 0,Y 140.059,Z 610.651,A -85,B 0,C 180,E1 -25802.13,E2 -25802.13} C_VEL
LIN {X 0,Y 138.13,Z 622.704,A -85,B 0,C 180,E1 -25803.773,E2 -25803.773} C_VEL
LIN {X 0,Y 135.561,Z 634.352,A -85,B 0,C 180,E1 -25805.91,E2 -25805.91} C_VEL
LIN {X 0,Y 132.493,Z 645.618,A -85,B 0,C 180,E1 -25808.618,E2 -25808.618} C_VEL
LIN {X 0,Y 129.329,Z 655.791,A -85,B 0,C 180,E1 -25811.798,E2 -25811.798} C_VEL
LIN {X 0,Y 126.104,Z 664.965,A -85,B 0,C 180,E1 -25815.481,E2 -25815.481} C_VEL
LIN {X 0,Y 122.795,Z 673.908,A -85,B 0,C 180,E1 -25820.119,E2 -25820.119} C_VEL
LIN {X 0,Y 119.872,Z 681.604,A -85,B 0,C 180,E1 -25825.324,E2 -25825.324} C_VEL
LIN {X 0,Y 117.963,Z 686.951,A -85,B 0,C 180,E1 -25830.006,E2 -25830.006} C_VEL
LIN {X 0,Y 116.551,Z 691.554,A -85,B 0,C 180,E1 -25835.195,E2 -25835.195} C_VEL
LIN {X 0,Y 115.952,Z 695.073,A -85,B 0,C 180,E1 -25840.482,E2 -25840.482} C_VEL
LIN {X 0,Y 115.996,Z 696.925,A -85,B 0,C 180,E1 -25844.212,E2 -25844.212} C_VEL
LIN {X 0,Y 117.081,Z 699.188,A -85,B 0,C 180,E1 -25851.116,E2 -25851.116} C_VEL
LIN {X 0,Y 119.665,Z 699.833,A -85,B 0,C 180,E1 -25858.03,E2 -25858.03} C_VEL
LIN {X 0,Y 121.513,Z 699.564,A -85,B 0,C 180,E1 -25861.374,E2 -25861.374} C_VEL
LIN {X 0,Y 123.719,Z 698.857,A -85,B 0,C 180,E1 -25864.622,E2 -25864.622} C_VEL
LIN {X 0,Y 128.08,Z 696.728,A -85,B 0,C 180,E1 -25869.809,E2 -25869.809} C_VEL
LIN {X 0,Y 132.207,Z 694.14,A -85,B 0,C 180,E1 -25873.721,E2 -25873.721} C_VEL
LIN {X 0,Y 132.448,Z 693.411,A -85,B 0,C 180,E1 -25875.122,E2 -25875.122} C_VEL
LIN {X 0,Y 123.324,Z 693.937,A -85,B 0,C 180,E1 -25881.182,E2 -25881.182} C_VEL
LIN {X 0,Y 116.455,Z 693.802,A -85,B 0,C 180,E1 -25888.635,E2 -25888.635} C_VEL
LIN {X 0,Y 116.25,Z 694.18,A -85,B 0,C 180,E1 -25889.457,E2 -25889.457} C_VEL
LIN {X 0,Y 114.644,Z 707.164,A -85,B 0,C 180,E1 -25894.59,E2 -25894.59} C_VEL
LIN {X 0,Y 113.732,Z 716.643,A -85,B 0,C 180,E1 -25899.189,E2 -25899.189} C_VEL
LIN {X 0,Y 113.143,Z 725.749,A -85,B 0,C 180,E1 -25904.694,E2 -25904.694} C_VEL
LIN {X 0,Y 113.093,Z 733.073,A -85,B 0,C 180,E1 -25910.162,E2 -25910.162} C_VEL
LIN {X 0,Y 114.014,Z 739.817,A -85,B 0,C 180,E1 -25916.467,E2 -25916.467} C_VEL
LIN {X 0,Y 116.49,Z 745.734,A -85,B 0,C 180,E1 -25923.46,E2 -25923.46} C_VEL
LIN {X 0,Y 120.805,Z 750.076,A -85,B 0,C 180,E1 -25930.053,E2 -25930.053} C_VEL
LIN {X 0,Y 126.781,Z 752.935,A -85,B 0,C 180,E1 -25936.093,E2 -25936.093} C_VEL
LIN {X 0,Y 134.354,Z 754.401,A -85,B 0,C 180,E1 -25941.481,E2 -25941.481} C_VEL
LIN {X 0,Y 143.144,Z 754.486,A -85,B 0,C 180,E1 -25946.225,E2 -25946.225} C_VEL
LIN {X 0,Y 153.149,Z 753.089,A -85,B 0,C 180,E1 -25950.318,E2 -25950.318} C_VEL
LIN {X 0,Y 158.417,Z 751.859,A -85,B 0,C 180,E1 -25952.167,E2 -25952.167} C_VEL
LIN {X 0,Y 169.763,Z 748.238,A -85,B 0,C 180,E1 -25955.422,E2 -25955.422} C_VEL
LIN {X 0,Y 176.058,Z 745.585,A -85,B 0,C 180,E1 -25957.019,E2 -25957.019} C_VEL
LIN {X 0,Y 164.452,Z 751.12,A -85,B 0,C 180,E1 -25959.708,E2 -25959.708} C_VEL
LIN {X 0,Y 153.536,Z 755.133,A -85,B 0,C 180,E1 -25962.907,E2 -25962.907} C_VEL
LIN {X 0,Y 143.556,Z 757.835,A -85,B 0,C 180,E1 -25966.728,E2 -25966.728} C_VEL
LIN {X 0,Y 134.626,Z 759.292,A -85,B 0,C 180,E1 -25971.206,E2 -25971.206} C_VEL
LIN {X 0,Y 127.153,Z 759.552,A -85,B 0,C 180,E1 -25976.44,E2 -25976.44} C_VEL
LIN {X 0,Y 126.438,Z 759.483,A -85,B 0,C 180,E1 -25977.047,E2 -25977.047} C_VEL
LIN {X 0,Y 123.262,Z 759.133,A -85,B 0,C 180,E1 -25979.319,E2 -25979.319} C_VEL
LIN {X 0,Y 117.061,Z 757.641,A -85,B 0,C 180,E1 -25982.931,E2 -25982.931} C_VEL
LIN {X 0,Y 111.569,Z 755.406,A -85,B 0,C 180,E1 -25986.913,E2 -25986.913} C_VEL
LIN {X 0,Y 109.617,Z 753.896,A -85,B 0,C 180,E1 -25989.702,E2 -25989.702} C_VEL
LIN {X 0,Y 108.151,Z 751.114,A -85,B 0,C 180,E1 -25994.928,E2 -25994.928} C_VEL
LIN {X 0,Y 107.943,Z 745.874,A -85,B 0,C 180,E1 -26002.512,E2 -26002.512} C_VEL
LIN {X 0,Y 108.446,Z 742.576,A -85,B 0,C 180,E1 -26006.278,E2 -26006.278} C_VEL
LIN {X 0,Y 108.484,Z 738.416,A -85,B 0,C 180,E1 -26009.994,E2 -26009.994} C_VEL
LIN {X 0,Y 108.246,Z 731.884,A -85,B 0,C 180,E1 -26014.649,E2 -26014.649} C_VEL
LIN {X 0,Y 108.356,Z 722.327,A -85,B 0,C 180,E1 -26020.268,E2 -26020.268} C_VEL
LIN {X 0,Y 108.527,Z 716.427,A -85,B 0,C 180,E1 -26026.936,E2 -26026.936} C_VEL
LIN {X 0,Y 110.046,Z 710.007,A -85,B 0,C 180,E1 -26032.524,E2 -26032.524} C_VEL
LIN {X 0,Y 112.683,Z 702.044,A -85,B 0,C 180,E1 -26037.883,E2 -26037.883} C_VEL
LIN {X 0,Y 115.668,Z 694.065,A -85,B 0,C 180,E1 -26042.027,E2 -26042.027} C_VEL
LIN {X 0,Y 119.477,Z 684.041,A -85,B 0,C 180,E1 -26046.024,E2 -26046.024} C_VEL
LIN {X 0,Y 123.434,Z 673.117,A -85,B 0,C 180,E1 -26049.296,E2 -26049.296} C_VEL
LIN {X 0,Y 126.775,Z 662.471,A -85,B 0,C 180,E1 -26051.693,E2 -26051.693} C_VEL
LIN {X 0,Y 130.062,Z 649.63,A -85,B 0,C 180,E1 -26053.807,E2 -26053.807} C_VEL
LIN {X 0,Y 132.485,Z 636.647,A -85,B 0,C 180,E1 -26055.334,E2 -26055.334} C_VEL
LIN {X 0,Y 134.044,Z 623.561,A -85,B 0,C 180,E1 -26056.315,E2 -26056.315} C_VEL
LIN {X 0,Y 134.48,Z 614.683,A -85,B 0,C 180,E1 -26056.82,E2 -26056.82} C_VEL
LIN {X 0,Y 133.429,Z 562.638,A -85,B 0,C 180,E1 -26060.917,E2 -26060.917} C_VEL
LIN {X 0,Y 129.163,Z 550.337,A -85,B 0,C 180,E1 -26063.719,E2 -26063.719} C_VEL
LIN {X 0,Y 124.697,Z 539.651,A -85,B 0,C 180,E1 -26066.846,E2 -26066.846} C_VEL
LIN {X 0,Y 121.402,Z 532.879,A -85,B 0,C 180,E1 -26069.324,E2 -26069.324} C_VEL
LIN {X 0,Y 118.846,Z 528.047,A -85,B 0,C 180,E1 -26071.403,E2 -26071.403} C_VEL
LIN {X 0,Y 115.883,Z 522.697,A -85,B 0,C 180,E1 -26074.035,E2 -26074.035} C_VEL
LIN {X 0,Y 112.225,Z 516.964,A -85,B 0,C 180,E1 -26077.668,E2 -26077.668} C_VEL
LIN {X 0,Y 109.151,Z 514.236,A -85,B 0,C 180,E1 -26080.975,E2 -26080.975} C_VEL
LIN {X 0,Y 108.046,Z 511.582,A -85,B 0,C 180,E1 -26082.978,E2 -26082.978} C_VEL
LIN {X 0,Y 107.994,Z 511.057,A -85,B 0,C 180,E1 -26084.427,E2 -26084.427} C_VEL
LIN {X 0,Y 108.277,Z 510.957,A -85,B 0,C 180,E1 -26088.77,E2 -26088.77} C_VEL
LIN {X 0,Y 108.443,Z 510.942,A -85,B 0,C 180,E1 -26096.283,E2 -26096.283} C_VEL
LIN {X 0,Y 108.909,Z 510.876,A -85,B 0,C 180,E1 -26099.999,E2 -26099.999} C_VEL
LIN {X 0,Y 108.31,Z 510.95,A -85,B 0,C 180,E1 -26107.455,E2 -26107.455} C_VEL
LIN {X 0,Y 108.185,Z 510.995,A -85,B 0,C 180,E1 -26113.013,E2 -26113.013} C_VEL
LIN {X 0,Y 107.896,Z 511,A -85,B 0,C 180,E1 -26119.006,E2 -26119.006} C_VEL
LIN {X 0,Y 107.846,Z 511.051,A -85,B 0,C 180,E1 -26124.186,E2 -26124.186} C_VEL
LIN {X 0,Y 107.796,Z 511.229,A -85,B 0,C 180,E1 -26132.481,E2 -26132.481} C_VEL
LIN {X 0,Y 107.972,Z 512.113,A -85,B 0,C 180,E1 -26133.726,E2 -26133.726} C_VEL
LIN {X 0,Y 109.291,Z 514.703,A -85,B 0,C 180,E1 -26135.634,E2 -26135.634} C_VEL
LIN {X 0,Y 112.245,Z 517.118,A -85,B 0,C 180,E1 -26138.764,E2 -26138.764} C_VEL
LIN {X 0,Y 114.233,Z 520.339,A -85,B 0,C 180,E1 -26140.818,E2 -26140.818} C_VEL
LIN {X 0,Y 116.127,Z 522.204,A -85,B 0,C 180,E1 -26142.489,E2 -26142.489} C_VEL
LIN {X 0,Y 118.651,Z 525.772,A -85,B 0,C 180,E1 -26144.649,E2 -26144.649} C_VEL
LIN {X 0,Y 123.013,Z 532.06,A -85,B 0,C 180,E1 -26147.962,E2 -26147.962} C_VEL
LIN {X 0,Y 127.952,Z 539.913,A -85,B 0,C 180,E1 -26151.263,E2 -26151.263} C_VEL
LIN {X 0,Y 133.092,Z 549.393,A -85,B 0,C 180,E1 -26154.351,E2 -26154.351} C_VEL
LIN {X 0,Y 137.797,Z 559.649,A -85,B 0,C 180,E1 -26156.963,E2 -26156.963} C_VEL
LIN {X 0,Y 135.899,Z 597.54,A -85,B 0,C 180,E1 -26159.01,E2 -26159.01} C_VEL
LIN {X 0,Y 134.47,Z 611.18,A -85,B 0,C 180,E1 -26160.318,E2 -26160.318} C_VEL
LIN {X 0,Y 132.29,Z 623.927,A -85,B 0,C 180,E1 -26162.091,E2 -26162.091} C_VEL
LIN {X 0,Y 129.615,Z 635.513,A -85,B 0,C 180,E1 -26164.299,E2 -26164.299} C_VEL
LIN {X 0,Y 126.378,Z 646.747,A -85,B 0,C 180,E1 -26167.096,E2 -26167.096} C_VEL
LIN {X 0,Y 123.011,Z 656.896,A -85,B 0,C 180,E1 -26170.394,E2 -26170.394} C_VEL
LIN {X 0,Y 119.28,Z 666.861,A -85,B 0,C 180,E1 -26174.631,E2 -26174.631} C_VEL
LIN {X 0,Y 115.815,Z 675.658,A -85,B 0,C 180,E1 -26179.517,E2 -26179.517} C_VEL
LIN {X 0,Y 112.921,Z 682.823,A -85,B 0,C 180,E1 -26184.738,E2 -26184.738} C_VEL
LIN {X 0,Y 110.823,Z 688.401,A -85,B 0,C 180,E1 -26190.006,E2 -26190.006} C_VEL
LIN {X 0,Y 109.418,Z 692.903,A -85,B 0,C 180,E1 -26195.535,E2 -26195.535} C_VEL
LIN {X 0,Y 108.888,Z 696.327,A -85,B 0,C 180,E1 -26201.171,E2 -26201.171} C_VEL
LIN {X 0,Y 109.005,Z 698.055,A -85,B 0,C 180,E1 -26204.951,E2 -26204.951} C_VEL
LIN {X 0,Y 109.476,Z 699.388,A -85,B 0,C 180,E1 -26208.729,E2 -26208.729} C_VEL
LIN {X 0,Y 110.346,Z 700.269,A -85,B 0,C 180,E1 -26212.473,E2 -26212.473} C_VEL
LIN {X 0,Y 113.31,Z 700.823,A -85,B 0,C 180,E1 -26219.755,E2 -26219.755} C_VEL
LIN {X 0,Y 115.381,Z 700.495,A -85,B 0,C 180,E1 -26223.25,E2 -26223.25} C_VEL
LIN {X 0,Y 117.79,Z 699.716,A -85,B 0,C 180,E1 -26226.638,E2 -26226.638} C_VEL
LIN {X 0,Y 122.197,Z 697.699,A -85,B 0,C 180,E1 -26231.612,E2 -26231.612} C_VEL
LIN {X 0,Y 124.474,Z 696.42,A -85,B 0,C 180,E1 -26233.778,E2 -26233.778} C_VEL
LIN {X 0,Y 123.929,Z 696.098,A -85,B 0,C 180,E1 -26235.17,E2 -26235.17} C_VEL
LIN {X 0,Y 114.795,Z 696.685,A -85,B 0,C 180,E1 -26242.251,E2 -26242.251} C_VEL
LIN {X 0,Y 108.893,Z 696.628,A -85,B 0,C 180,E1 -26249.989,E2 -26249.989} C_VEL
LIN {X 0,Y 108.785,Z 696.988,A -85,B 0,C 180,E1 -26250.887,E2 -26250.887} C_VEL
LIN {X 0,Y 107.171,Z 711.223,A -85,B 0,C 180,E1 -26257.322,E2 -26257.322} C_VEL
LIN {X 0,Y 106.375,Z 720.773,A -85,B 0,C 180,E1 -26262.706,E2 -26262.706} C_VEL
LIN {X 0,Y 106.148,Z 727.774,A -85,B 0,C 180,E1 -26267.575,E2 -26267.575} C_VEL
LIN {X 0,Y 106.502,Z 734.919,A -85,B 0,C 180,E1 -26273.636,E2 -26273.636} C_VEL
LIN {X 0,Y 107.982,Z 741.107,A -85,B 0,C 180,E1 -26280.001,E2 -26280.001} C_VEL
LIN {X 0,Y 111.311,Z 746.769,A -85,B 0,C 180,E1 -26287.256,E2 -26287.256} C_VEL
LIN {X 0,Y 116.605,Z 750.953,A -85,B 0,C 180,E1 -26293.952,E2 -26293.952} C_VEL
LIN {X 0,Y 123.521,Z 753.669,A -85,B 0,C 180,E1 -26299.962,E2 -26299.962} C_VEL
LIN {X 0,Y 132.209,Z 755.081,A -85,B 0,C 180,E1 -26305.342,E2 -26305.342} C_VEL
LIN {X 0,Y 141.678,Z 755.034,A -85,B 0,C 180,E1 -26309.74,E2 -26309.74} C_VEL
LIN {X 0,Y 152.385,Z 753.585,A -85,B 0,C 180,E1 -26313.605,E2 -26313.605} C_VEL
LIN {X 0,Y 162.27,Z 751.168,A -85,B 0,C 180,E1 -26316.447,E2 -26316.447} C_VEL
LIN {X 0,Y 162.442,Z 751.231,A -85,B 0,C 180,E1 -26317.198,E2 -26317.198} C_VEL
LIN {X 0,Y 154.316,Z 754.08,A -85,B 0,C 180,E1 -26319.259,E2 -26319.259} C_VEL
LIN {X 0,Y 143.514,Z 756.918,A -85,B 0,C 180,E1 -26322.723,E2 -26322.723} C_VEL
LIN {X 0,Y 133.739,Z 758.537,A -85,B 0,C 180,E1 -26326.903,E2 -26326.903} C_VEL
LIN {X 0,Y 125.04,Z 758.954,A -85,B 0,C 180,E1 -26331.804,E2 -26331.804} C_VEL
LIN {X 0,Y 117.952,Z 758.226,A -85,B 0,C 180,E1 -26337.565,E2 -26337.565} C_VEL
LIN {X 0,Y 112.462,Z 756.295,A -85,B 0,C 180,E1 -26344.053,E2 -26344.053} C_VEL
LIN {X 0,Y 109.617,Z 753.896,A -85,B 0,C 180,E1 -26349.702,E2 -26349.702} C_VEL
LIN {X 0,Y 108.065,Z 752.254,A -85,B 0,C 180,E1 -26352.564,E2 -26352.564} C_VEL
LIN {X 0,Y 104.664,Z 748.476,A -85,B 0,C 180,E1 -26357.137,E2 -26357.137} C_VEL
LIN {X 0,Y 101.983,Z 743.946,A -85,B 0,C 180,E1 -26361.836,E2 -26361.836} C_VEL
LIN {X 0,Y 101.635,Z 741.134,A -85,B 0,C 180,E1 -26364.795,E2 -26364.795} C_VEL
LIN {X 0,Y 101.839,Z 737.95,A -85,B 0,C 180,E1 -26368.016,E2 -26368.016} C_VEL
LIN {X 0,Y 101.549,Z 731.571,A -85,B 0,C 180,E1 -26372.969,E2 -26372.969} C_VEL
LIN {X 0,Y 101.424,Z 722.616,A -85,B 0,C 180,E1 -26378.712,E2 -26378.712} C_VEL
LIN {X 0,Y 101.33,Z 716.908,A -85,B 0,C 180,E1 -26386.1,E2 -26386.1} C_VEL
LIN {X 0,Y 102.676,Z 710.819,A -85,B 0,C 180,E1 -26392.108,E2 -26392.108} C_VEL
LIN {X 0,Y 105.24,Z 703.25,A -85,B 0,C 180,E1 -26397.862,E2 -26397.862} C_VEL
LIN {X 0,Y 109.042,Z 693.816,A -85,B 0,C 180,E1 -26403.281,E2 -26403.281} C_VEL
LIN {X 0,Y 112.916,Z 684.264,A -85,B 0,C 180,E1 -26407.354,E2 -26407.354} C_VEL
LIN {X 0,Y 117.024,Z 673.581,A -85,B 0,C 180,E1 -26410.768,E2 -26410.768} C_VEL
LIN {X 0,Y 121.011,Z 661.666,A -85,B 0,C 180,E1 -26413.596,E2 -26413.596} C_VEL
LIN {X 0,Y 124.189,Z 650.026,A -85,B 0,C 180,E1 -26415.591,E2 -26415.591} C_VEL
LIN {X 0,Y 126.872,Z 636.626,A -85,B 0,C 180,E1 -26417.247,E2 -26417.247} C_VEL
LIN {X 0,Y 128.584,Z 623.543,A -85,B 0,C 180,E1 -26418.296,E2 -26418.296} C_VEL
LIN {X 0,Y 129.037,Z 615.468,A -85,B 0,C 180,E1 -26418.778,E2 -26418.778} C_VEL
LIN {X 0,Y 128.326,Z 564.754,A -85,B 0,C 180,E1 -26422.954,E2 -26422.954} C_VEL
LIN {X 0,Y 124.207,Z 552.649,A -85,B 0,C 180,E1 -26425.968,E2 -26425.968} C_VEL
LIN {X 0,Y 119.628,Z 541.663,A -85,B 0,C 180,E1 -26429.554,E2 -26429.554} C_VEL
LIN {X 0,Y 115.768,Z 533.619,A -85,B 0,C 180,E1 -26432.914,E2 -26432.914} C_VEL
LIN {X 0,Y 112.824,Z 528.075,A -85,B 0,C 180,E1 -26435.783,E2 -26435.783} C_VEL
LIN {X 0,Y 109.555,Z 522.915,A -85,B 0,C 180,E1 -26439.338,E2 -26439.338} C_VEL
LIN {X 0,Y 107.107,Z 520.65,A -85,B 0,C 180,E1 -26442.209,E2 -26442.209} C_VEL
LIN {X 0,Y 105.54,Z 517.715,A -85,B 0,C 180,E1 -26444.551,E2 -26444.551} C_VEL
LIN {X 0,Y 102.898,Z 515.597,A -85,B 0,C 180,E1 -26448.674,E2 -26448.674} C_VEL
LIN {X 0,Y 101.51,Z 513.113,A -85,B 0,C 180,E1 -26451.789,E2 -26451.789} C_VEL
LIN {X 0,Y 101.325,Z 512.127,A -85,B 0,C 180,E1 -26453.777,E2 -26453.777} C_VEL
LIN {X 0,Y 101.837,Z 511.755,A -85,B 0,C 180,E1 -26459.999,E2 -26459.999} C_VEL
LIN {X 0,Y 101.25,Z 511.825,A -85,B 0,C 180,E1 -26467.978,E2 -26467.978} C_VEL
LIN {X 0,Y 101.111,Z 511.878,A -85,B 0,C 180,E1 -26473.349,E2 -26473.349} C_VEL
LIN {X 0,Y 100.806,Z 511.958,A -85,B 0,C 180,E1 -26480.399,E2 -26480.399} C_VEL
LIN {X 0,Y 100.995,Z 512.731,A -85,B 0,C 180,E1 -26483.313,E2 -26483.313} C_VEL
LIN {X 0,Y 102.199,Z 515.476,A -85,B 0,C 180,E1 -26486.551,E2 -26486.551} C_VEL
LIN {X 0,Y 104.765,Z 517.513,A -85,B 0,C 180,E1 -26490.829,E2 -26490.829} C_VEL
LIN {X 0,Y 105.621,Z 518.096,A -85,B 0,C 180,E1 -26492.037,E2 -26492.037} C_VEL
LIN {X 0,Y 107.151,Z 520.976,A -85,B 0,C 180,E1 -26494.308,E2 -26494.308} C_VEL
LIN {X 0,Y 109.803,Z 523.352,A -85,B 0,C 180,E1 -26497.366,E2 -26497.366} C_VEL
LIN {X 0,Y 111.978,Z 526.743,A -85,B 0,C 180,E1 -26499.745,E2 -26499.745} C_VEL
LIN {X 0,Y 113.676,Z 528.703,A -85,B 0,C 180,E1 -26501.356,E2 -26501.356} C_VEL
LIN {X 0,Y 116.937,Z 533.357,A -85,B 0,C 180,E1 -26504.274,E2 -26504.274} C_VEL
LIN {X 0,Y 121.368,Z 540.122,A -85,B 0,C 180,E1 -26507.757,E2 -26507.757} C_VEL
LIN {X 0,Y 126.165,Z 548.562,A -85,B 0,C 180,E1 -26511.1,E2 -26511.1} C_VEL
LIN {X 0,Y 130.796,Z 558.134,A -85,B 0,C 180,E1 -26514.03,E2 -26514.03} C_VEL
LIN {X 0,Y 132.45,Z 562.023,A -85,B 0,C 180,E1 -26515.029,E2 -26515.029} C_VEL
LIN {X 0,Y 130.492,Z 598.443,A -85,B 0,C 180,E1 -26517.061,E2 -26517.061} C_VEL
LIN {X 0,Y 129.017,Z 611.795,A -85,B 0,C 180,E1 -26518.371,E2 -26518.371} C_VEL
LIN {X 0,Y 126.834,Z 624.085,A -85,B 0,C 180,E1 -26520.092,E2 -26520.092} C_VEL
LIN {X 0,Y 124.201,Z 635.078,A -85,B 0,C 180,E1 -26522.178,E2 -26522.178} C_VEL
LIN {X 0,Y 120.736,Z 646.575,A -85,B 0,C 180,E1 -26525.044,E2 -26525.044} C_VEL
LIN {X 0,Y 117.175,Z 656.923,A -85,B 0,C 180,E1 -26528.453,E2 -26528.453} C_VEL
LIN {X 0,Y 113.833,Z 665.435,A -85,B 0,C 180,E1 -26532.026,E2 -26532.026} C_VEL
LIN {X 0,Y 110.6,Z 673.284,A -85,B 0,C 180,E1 -26536.221,E2 -26536.221} C_VEL
LIN {X 0,Y 107.211,Z 681.001,A -85,B 0,C 180,E1 -26541.525,E2 -26541.525} C_VEL
LIN {X 0,Y 105.047,Z 686.289,A -85,B 0,C 180,E1 -26546.17,E2 -26546.17} C_VEL
LIN {X 0,Y 103.117,Z 691.446,A -85,B 0,C 180,E1 -26551.959,E2 -26551.959} C_VEL
LIN {X 0,Y 102.018,Z 695.484,A -85,B 0,C 180,E1 -26557.926,E2 -26557.926} C_VEL
LIN {X 0,Y 101.97,Z 698.966,A -85,B 0,C 180,E1 -26565.23,E2 -26565.23} C_VEL
LIN {X 0,Y 102.655,Z 700.523,A -85,B 0,C 180,E1 -26570.025,E2 -26570.025} C_VEL
LIN {X 0,Y 105.165,Z 701.776,A -85,B 0,C 180,E1 -26577.898,E2 -26577.898} C_VEL
LIN {X 0,Y 107.065,Z 701.813,A -85,B 0,C 180,E1 -26581.685,E2 -26581.685} C_VEL
LIN {X 0,Y 109.376,Z 701.398,A -85,B 0,C 180,E1 -26585.338,E2 -26585.338} C_VEL
LIN {X 0,Y 112.042,Z 700.572,A -85,B 0,C 180,E1 -26588.856,E2 -26588.856} C_VEL
LIN {X 0,Y 116.413,Z 698.683,A -85,B 0,C 180,E1 -26593.578,E2 -26593.578} C_VEL
LIN {X 0,Y 113.144,Z 698.774,A -85,B 0,C 180,E1 -26596.902,E2 -26596.902} C_VEL
LIN {X 0,Y 103.63,Z 699.352,A -85,B 0,C 180,E1 -26607.145,E2 -26607.145} C_VEL
LIN {X 0,Y 101.327,Z 699.36,A -85,B 0,C 180,E1 -26612.198,E2 -26612.198} C_VEL
LIN {X 0,Y 101.281,Z 699.927,A -85,B 0,C 180,E1 -26612.8,E2 -26612.8} C_VEL
LIN {X 0,Y 100.075,Z 711.514,A -85,B 0,C 180,E1 -26618.496,E2 -26618.496} C_VEL
LIN {X 0,Y 99.415,Z 721.447,A -85,B 0,C 180,E1 -26624.629,E2 -26624.629} C_VEL
LIN {X 0,Y 99.387,Z 729.629,A -85,B 0,C 180,E1 -26630.95,E2 -26630.95} C_VEL
LIN {X 0,Y 100.404,Z 737.051,A -85,B 0,C 180,E1 -26637.996,E2 -26637.996} C_VEL
LIN {X 0,Y 102.341,Z 742.226,A -85,B 0,C 180,E1 -26643.939,E2 -26643.939} C_VEL
LIN {X 0,Y 106.689,Z 747.765,A -85,B 0,C 180,E1 -26651.399,E2 -26651.399} C_VEL
LIN {X 0,Y 112.988,Z 751.75,A -85,B 0,C 180,E1 -26658.121,E2 -26658.121} C_VEL
LIN {X 0,Y 120.927,Z 754.396,A -85,B 0,C 180,E1 -26664.007,E2 -26664.007} C_VEL
LIN {X 0,Y 130.244,Z 755.705,A -85,B 0,C 180,E1 -26669.056,E2 -26669.056} C_VEL
LIN {X 0,Y 140.805,Z 755.595,A -85,B 0,C 180,E1 -26673.303,E2 -26673.303} C_VEL
LIN {X 0,Y 150.261,Z 754.455,A -85,B 0,C 180,E1 -26676.332,E2 -26676.332} C_VEL
LIN {X 0,Y 149.943,Z 754.661,A -85,B 0,C 180,E1 -26677.167,E2 -26677.167} C_VEL
LIN {X 0,Y 138.804,Z 757.048,A -85,B 0,C 180,E1 -26680.574,E2 -26680.574} C_VEL
LIN {X 0,Y 128.667,Z 758.217,A -85,B 0,C 180,E1 -26684.752,E2 -26684.752} C_VEL
LIN {X 0,Y 119.567,Z 758.21,A -85,B 0,C 180,E1 -26689.71,E2 -26689.71} C_VEL
LIN {X 0,Y 112.098,Z 757.088,A -85,B 0,C 180,E1 -26695.643,E2 -26695.643} C_VEL
LIN {X 0,Y 106.253,Z 754.809,A -85,B 0,C 180,E1 -26702.412,E2 -26702.412} C_VEL
LIN {X 0,Y 102.612,Z 751.309,A -85,B 0,C 180,E1 -26709.967,E2 -26709.967} C_VEL
LIN {X 0,Y 101.19,Z 746.503,A -85,B 0,C 180,E1 -26717.967,E2 -26717.967} C_VEL
LIN {X 0,Y 101.635,Z 741.134,A -85,B 0,C 180,E1 -26724.795,E2 -26724.795} C_VEL
LIN {X 0,Y 101.151,Z 739.104,A -85,B 0,C 180,E1 -26726.635,E2 -26726.635} C_VEL
LIN {X 0,Y 99.717,Z 736.714,A -85,B 0,C 180,E1 -26728.248,E2 -26728.248} C_VEL
LIN {X 0,Y 95.58,Z 730.45,A -85,B 0,C 180,E1 -26731.79,E2 -26731.79} C_VEL
LIN {X 0,Y 94.771,Z 727.645,A -85,B 0,C 180,E1 -26733.552,E2 -26733.552} C_VEL
LIN {X 0,Y 94.589,Z 722.728,A -85,B 0,C 180,E1 -26736.927,E2 -26736.927} C_VEL
LIN {X 0,Y 94.104,Z 718.236,A -85,B 0,C 180,E1 -26743.853,E2 -26743.853} C_VEL
LIN {X 0,Y 95.041,Z 712.566,A -85,B 0,C 180,E1 -26750.556,E2 -26750.556} C_VEL
LIN {X 0,Y 97.349,Z 705.675,A -85,B 0,C 180,E1 -26756.814,E2 -26756.814} C_VEL
LIN {X 0,Y 100.862,Z 697.159,A -85,B 0,C 180,E1 -26762.676,E2 -26762.676} C_VEL
LIN {X 0,Y 104.654,Z 688.455,A -85,B 0,C 180,E1 -26767.177,E2 -26767.177} C_VEL
LIN {X 0,Y 109.246,Z 677.761,A -85,B 0,C 180,E1 -26771.246,E2 -26771.246} C_VEL
LIN {X 0,Y 113.268,Z 667.155,A -85,B 0,C 180,E1 -26774.261,E2 -26774.261} C_VEL
LIN {X 0,Y 117.062,Z 655.476,A -85,B 0,C 180,E1 -26776.705,E2 -26776.705} C_VEL
LIN {X 0,Y 120.131,Z 643.294,A -85,B 0,C 180,E1 -26778.544,E2 -26778.544} C_VEL
LIN {X 0,Y 122.429,Z 630.151,A -85,B 0,C 180,E1 -26779.955,E2 -26779.955} C_VEL
LIN {X 0,Y 123.787,Z 617.24,A -85,B 0,C 180,E1 -26780.816,E2 -26780.816} C_VEL
LIN {X 0,Y 123.416,Z 567.101,A -85,B 0,C 180,E1 -26785.128,E2 -26785.128} C_VEL
LIN {X 0,Y 120.011,Z 556.615,A -85,B 0,C 180,E1 -26787.914,E2 -26787.914} C_VEL
LIN {X 0,Y 115.802,Z 546.001,A -85,B 0,C 180,E1 -26791.572,E2 -26791.572} C_VEL
LIN {X 0,Y 112.44,Z 538.665,A -85,B 0,C 180,E1 -26794.829,E2 -26794.829} C_VEL
LIN {X 0,Y 109.832,Z 533.428,A -85,B 0,C 180,E1 -26797.669,E2 -26797.669} C_VEL
LIN {X 0,Y 107.155,Z 529.218,A -85,B 0,C 180,E1 -26800.855,E2 -26800.855} C_VEL
LIN {X 0,Y 104.665,Z 526.326,A -85,B 0,C 180,E1 -26804.168,E2 -26804.168} C_VEL
LIN {X 0,Y 103.751,Z 524.389,A -85,B 0,C 180,E1 -26805.707,E2 -26805.707} C_VEL
LIN {X 0,Y 100.903,Z 521.648,A -85,B 0,C 180,E1 -26810.73,E2 -26810.73} C_VEL
LIN {X 0,Y 99.666,Z 519.064,A -85,B 0,C 180,E1 -26813.927,E2 -26813.927} C_VEL
LIN {X 0,Y 97.795,Z 517.612,A -85,B 0,C 180,E1 -26819.998,E2 -26819.998} C_VEL
LIN {X 0,Y 96.894,Z 517.502,A -85,B 0,C 180,E1 -26830.446,E2 -26830.446} C_VEL
LIN {X 0,Y 99.347,Z 519.161,A -85,B 0,C 180,E1 -26841.752,E2 -26841.752} C_VEL
LIN {X 0,Y 100.842,Z 522.32,A -85,B 0,C 180,E1 -26845.76,E2 -26845.76} C_VEL
LIN {X 0,Y 103.339,Z 524.363,A -85,B 0,C 180,E1 -26850.169,E2 -26850.169} C_VEL
LIN {X 0,Y 103.842,Z 525.119,A -85,B 0,C 180,E1 -26850.995,E2 -26850.995} C_VEL
LIN {X 0,Y 105.904,Z 528.265,A -85,B 0,C 180,E1 -26854.049,E2 -26854.049} C_VEL
LIN {X 0,Y 107.618,Z 529.932,A -85,B 0,C 180,E1 -26856.135,E2 -26856.135} C_VEL
LIN {X 0,Y 110.185,Z 533.584,A -85,B 0,C 180,E1 -26859.055,E2 -26859.055} C_VEL
LIN {X 0,Y 114.131,Z 539.32,A -85,B 0,C 180,E1 -26862.913,E2 -26862.913} C_VEL
LIN {X 0,Y 118.17,Z 545.849,A -85,B 0,C 180,E1 -26866.364,E2 -26866.364} C_VEL
LIN {X 0,Y 122.443,Z 553.726,A -85,B 0,C 180,E1 -26869.607,E2 -26869.607} C_VEL
LIN {X 0,Y 126.615,Z 562.754,A -85,B 0,C 180,E1 -26872.496,E2 -26872.496} C_VEL
LIN {X 0,Y 127.286,Z 564.32,A -85,B 0,C 180,E1 -26872.938,E2 -26872.938} C_VEL
LIN {X 0,Y 125.241,Z 599.453,A -85,B 0,C 180,E1 -26874.956,E2 -26874.956} C_VEL
LIN {X 0,Y 123.6,Z 613.156,A -85,B 0,C 180,E1 -26876.338,E2 -26876.338} C_VEL
LIN {X 0,Y 121.311,Z 625.259,A -85,B 0,C 180,E1 -26878.093,E2 -26878.093} C_VEL
LIN {X 0,Y 118.05,Z 637.769,A -85,B 0,C 180,E1 -26880.59,E2 -26880.59} C_VEL
LIN {X 0,Y 114.412,Z 648.954,A -85,B 0,C 180,E1 -26883.561,E2 -26883.561} C_VEL
LIN {X 0,Y 110.638,Z 659.042,A -85,B 0,C 180,E1 -26887.11,E2 -26887.11} C_VEL
LIN {X 0,Y 106.415,Z 668.977,A -85,B 0,C 180,E1 -26891.724,E2 -26891.724} C_VEL
LIN {X 0,Y 102.492,Z 677.749,A -85,B 0,C 180,E1 -26897.13,E2 -26897.13} C_VEL
LIN {X 0,Y 99.064,Z 685.22,A -85,B 0,C 180,E1 -26903.31,E2 -26903.31} C_VEL
LIN {X 0,Y 96.526,Z 691.281,A -85,B 0,C 180,E1 -26910.007,E2 -26910.007} C_VEL
LIN {X 0,Y 95.148,Z 695.589,A -85,B 0,C 180,E1 -26916.368,E2 -26916.368} C_VEL
LIN {X 0,Y 94.824,Z 698.826,A -85,B 0,C 180,E1 -26922.854,E2 -26922.854} C_VEL
LIN {X 0,Y 95.118,Z 700.468,A -85,B 0,C 180,E1 -26927.198,E2 -26927.198} C_VEL
LIN {X 0,Y 95.889,Z 701.643,A -85,B 0,C 180,E1 -26931.505,E2 -26931.505} C_VEL
LIN {X 0,Y 98.829,Z 702.809,A -85,B 0,C 180,E1 -26939.861,E2 -26939.861} C_VEL
LIN {X 0,Y 100.961,Z 702.773,A -85,B 0,C 180,E1 -26943.848,E2 -26943.848} C_VEL
LIN {X 0,Y 106.475,Z 701.431,A -85,B 0,C 180,E1 -26951.313,E2 -26951.313} C_VEL
LIN {X 0,Y 108.005,Z 700.652,A -85,B 0,C 180,E1 -26954.295,E2 -26954.295} C_VEL
LIN {X 0,Y 97.915,Z 701.647,A -85,B 0,C 180,E1 -26964.957,E2 -26964.957} C_VEL
LIN {X 0,Y 93.916,Z 701.819,A -85,B 0,C 180,E1 -26974.094,E2 -26974.094} C_VEL
LIN {X 0,Y 93.857,Z 702.694,A -85,B 0,C 180,E1 -26975.004,E2 -26975.004} C_VEL
LIN {X 0,Y 92.885,Z 713.879,A -85,B 0,C 180,E1 -26981.244,E2 -26981.244} C_VEL
LIN {X 0,Y 92.522,Z 723.466,A -85,B 0,C 180,E1 -26987.945,E2 -26987.945} C_VEL
LIN {X 0,Y 92.821,Z 730.596,A -85,B 0,C 180,E1 -26994.116,E2 -26994.116} C_VEL
LIN {X 0,Y 94.586,Z 738.296,A -85,B 0,C 180,E1 -27002.131,E2 -27002.131} C_VEL
LIN {X 0,Y 97.241,Z 743.31,A -85,B 0,C 180,E1 -27008.313,E2 -27008.313} C_VEL
LIN {X 0,Y 102.683,Z 748.627,A -85,B 0,C 180,E1 -27015.89,E2 -27015.89} C_VEL
LIN {X 0,Y 110.007,Z 752.522,A -85,B 0,C 180,E1 -27022.541,E2 -27022.541} C_VEL
LIN {X 0,Y 118.979,Z 755.097,A -85,B 0,C 180,E1 -27028.202,E2 -27028.202} C_VEL
LIN {X 0,Y 129.181,Z 756.334,A -85,B 0,C 180,E1 -27032.961,E2 -27032.961} C_VEL
LIN {X 0,Y 138.367,Z 756.326,A -85,B 0,C 180,E1 -27036.216,E2 -27036.216} C_VEL
LIN {X 0,Y 136.606,Z 756.685,A -85,B 0,C 180,E1 -27037.545,E2 -27037.545} C_VEL
LIN {X 0,Y 128.891,Z 757.489,A -85,B 0,C 180,E1 -27040.23,E2 -27040.23} C_VEL
LIN {X 0,Y 118.843,Z 757.646,A -85,B 0,C 180,E1 -27044.787,E2 -27044.787} C_VEL
LIN {X 0,Y 110.147,Z 756.699,A -85,B 0,C 180,E1 -27050.346,E2 -27050.346} C_VEL
LIN {X 0,Y 103.054,Z 754.628,A -85,B 0,C 180,E1 -27056.928,E2 -27056.928} C_VEL
LIN {X 0,Y 97.942,Z 751.414,A -85,B 0,C 180,E1 -27064.491,E2 -27064.491} C_VEL
LIN {X 0,Y 95.104,Z 746.874,A -85,B 0,C 180,E1 -27072.8,E2 -27072.8} C_VEL
LIN {X 0,Y 94.758,Z 740.98,A -85,B 0,C 180,E1 -27081.462,E2 -27081.462} C_VEL
LIN {X 0,Y 95.261,Z 736.157,A -85,B 0,C 180,E1 -27086.821,E2 -27086.821} C_VEL
LIN {X 0,Y 94.862,Z 729.656,A -85,B 0,C 180,E1 -27092.116,E2 -27092.116} C_VEL
LIN {X 0,Y 94.771,Z 727.645,A -85,B 0,C 180,E1 -27093.552,E2 -27093.552} C_VEL
LIN {X 0,Y 94.27,Z 725.25,A -85,B 0,C 180,E1 -27095.381,E2 -27095.381} C_VEL
LIN {X 0,Y 93.268,Z 723.169,A -85,B 0,C 180,E1 -27097.3,E2 -27097.3} C_VEL
LIN {X 0,Y 90.613,Z 719.621,A -85,B 0,C 180,E1 -27101.375,E2 -27101.375} C_VEL
LIN {X 0,Y 87.958,Z 715.443,A -85,B 0,C 180,E1 -27107.01,E2 -27107.01} C_VEL
LIN {X 0,Y 87.89,Z 712.609,A -85,B 0,C 180,E1 -27110.502,E2 -27110.502} C_VEL
LIN {X 0,Y 90.434,Z 705.387,A -85,B 0,C 180,E1 -27117.785,E2 -27117.785} C_VEL
LIN {X 0,Y 94.17,Z 697.019,A -85,B 0,C 180,E1 -27124.028,E2 -27124.028} C_VEL
LIN {X 0,Y 98.548,Z 687.667,A -85,B 0,C 180,E1 -27129.191,E2 -27129.191} C_VEL
LIN {X 0,Y 103.449,Z 676.896,A -85,B 0,C 180,E1 -27133.451,E2 -27133.451} C_VEL
LIN {X 0,Y 107.72,Z 666.325,A -85,B 0,C 180,E1 -27136.529,E2 -27136.529} C_VEL
LIN {X 0,Y 111.692,Z 654.689,A -85,B 0,C 180,E1 -27139.022,E2 -27139.022} C_VEL
LIN {X 0,Y 114.902,Z 642.568,A -85,B 0,C 180,E1 -27140.889,E2 -27140.889} C_VEL
LIN {X 0,Y 117.434,Z 628.855,A -85,B 0,C 180,E1 -27142.372,E2 -27142.372} C_VEL
LIN {X 0,Y 118.685,Z 617.758,A -85,B 0,C 180,E1 -27143.134,E2 -27143.134} C_VEL
LIN {X 0,Y 118.658,Z 569.351,A -85,B 0,C 180,E1 -27147.503,E2 -27147.503} C_VEL
LIN {X 0,Y 115.732,Z 559.96,A -85,B 0,C 180,E1 -27150.184,E2 -27150.184} C_VEL
LIN {X 0,Y 111.684,Z 549.155,A -85,B 0,C 180,E1 -27154.2,E2 -27154.2} C_VEL
LIN {X 0,Y 109.04,Z 543.211,A -85,B 0,C 180,E1 -27157.11,E2 -27157.11} C_VEL
LIN {X 0,Y 106.862,Z 538.533,A -85,B 0,C 180,E1 -27159.8,E2 -27159.8} C_VEL
LIN {X 0,Y 105.02,Z 535.557,A -85,B 0,C 180,E1 -27162.221,E2 -27162.221} C_VEL
LIN {X 0,Y 102.604,Z 532.435,A -85,B 0,C 180,E1 -27165.783,E2 -27165.783} C_VEL
LIN {X 0,Y 101.649,Z 530.767,A -85,B 0,C 180,E1 -27167.495,E2 -27167.495} C_VEL
LIN {X 0,Y 98.953,Z 527.423,A -85,B 0,C 180,E1 -27173.114,E2 -27173.114} C_VEL
LIN {X 0,Y 98.258,Z 525.776,A -85,B 0,C 180,E1 -27175.245,E2 -27175.245} C_VEL
LIN {X 0,Y 96.889,Z 524.717,A -85,B 0,C 180,E1 -27179.998,E2 -27179.998} C_VEL
LIN {X 0,Y 96.011,Z 524.562,A -85,B 0,C 180,E1 -27190.543,E2 -27190.543} C_VEL
LIN {X 0,Y 98.054,Z 526.042,A -85,B 0,C 180,E1 -27200.724,E2 -27200.724} C_VEL
LIN {X 0,Y 99.435,Z 529.047,A -85,B 0,C 180,E1 -27204.769,E2 -27204.769} C_VEL
LIN {X 0,Y 101.917,Z 531.46,A -85,B 0,C 180,E1 -27209.494,E2 -27209.494} C_VEL
LIN {X 0,Y 104.087,Z 534.843,A -85,B 0,C 180,E1 -27212.981,E2 -27212.981} C_VEL
LIN {X 0,Y 105.537,Z 536.481,A -85,B 0,C 180,E1 -27214.908,E2 -27214.908} C_VEL
LIN {X 0,Y 108.783,Z 541.223,A -85,B 0,C 180,E1 -27218.789,E2 -27218.789} C_VEL
LIN {X 0,Y 112.624,Z 547.222,A -85,B 0,C 180,E1 -27222.672,E2 -27222.672} C_VEL
LIN {X 0,Y 117.429,Z 555.951,A -85,B 0,C 180,E1 -27226.899,E2 -27226.899} C_VEL
LIN {X 0,Y 121.867,Z 565.643,A -85,B 0,C 180,E1 -27230.357,E2 -27230.357} C_VEL
LIN {X 0,Y 122.366,Z 567.317,A -85,B 0,C 180,E1 -27230.767,E2 -27230.767} C_VEL
LIN {X 0,Y 120.159,Z 600.546,A -85,B 0,C 180,E1 -27232.675,E2 -27232.675} C_VEL
LIN {X 0,Y 118.485,Z 613.689,A -85,B 0,C 180,E1 -27234.021,E2 -27234.021} C_VEL
LIN {X 0,Y 115.932,Z 626.437,A -85,B 0,C 180,E1 -27235.9,E2 -27235.9} C_VEL
LIN {X 0,Y 112.481,Z 638.898,A -85,B 0,C 180,E1 -27238.455,E2 -27238.455} C_VEL
LIN {X 0,Y 108.638,Z 650.05,A -85,B 0,C 180,E1 -27241.511,E2 -27241.511} C_VEL
LIN {X 0,Y 104.601,Z 660.117,A -85,B 0,C 180,E1 -27245.177,E2 -27245.177} C_VEL
LIN {X 0,Y 100.483,Z 669.224,A -85,B 0,C 180,E1 -27249.538,E2 -27249.538} C_VEL
LIN {X 0,Y 96.236,Z 678.117,A -85,B 0,C 180,E1 -27255.198,E2 -27255.198} C_VEL
LIN {X 0,Y 92.688,Z 685.31,A -85,B 0,C 180,E1 -27261.285,E2 -27261.285} C_VEL
LIN {X 0,Y 90.05,Z 691.064,A -85,B 0,C 180,E1 -27267.771,E2 -27267.771} C_VEL
LIN {X 0,Y 88.353,Z 695.637,A -85,B 0,C 180,E1 -27274.57,E2 -27274.57} C_VEL
LIN {X 0,Y 87.785,Z 699.126,A -85,B 0,C 180,E1 -27281.553,E2 -27281.553} C_VEL
LIN {X 0,Y 88.246,Z 701.636,A -85,B 0,C 180,E1 -27288.584,E2 -27288.584} C_VEL
LIN {X 0,Y 90.669,Z 703.498,A -85,B 0,C 180,E1 -27297.723,E2 -27297.723} C_VEL
LIN {X 0,Y 94.068,Z 703.81,A -85,B 0,C 180,E1 -27304.734,E2 -27304.734} C_VEL
LIN {X 0,Y 99.394,Z 702.818,A -85,B 0,C 180,E1 -27312.1,E2 -27312.1} C_VEL
LIN {X 0,Y 100.129,Z 702.5,A -85,B 0,C 180,E1 -27314.012,E2 -27314.012} C_VEL
LIN {X 0,Y 89.685,Z 703.83,A -85,B 0,C 180,E1 -27326.735,E2 -27326.735} C_VEL
LIN {X 0,Y 86.581,Z 704.177,A -85,B 0,C 180,E1 -27336.691,E2 -27336.691} C_VEL
LIN {X 0,Y 86.542,Z 705.277,A -85,B 0,C 180,E1 -27337.627,E2 -27337.627} C_VEL
LIN {X 0,Y 85.9,Z 714.547,A -85,B 0,C 180,E1 -27343.362,E2 -27343.362} C_VEL
LIN {X 0,Y 85.811,Z 723.833,A -85,B 0,C 180,E1 -27350.574,E2 -27350.574} C_VEL
LIN {X 0,Y 86.736,Z 732.48,A -85,B 0,C 180,E1 -27358.841,E2 -27358.841} C_VEL
LIN {X 0,Y 89.294,Z 739.398,A -85,B 0,C 180,E1 -27366.782,E2 -27366.782} C_VEL
LIN {X 0,Y 94.28,Z 745.695,A -85,B 0,C 180,E1 -27375.127,E2 -27375.127} C_VEL
LIN {X 0,Y 101.354,Z 750.541,A -85,B 0,C 180,E1 -27382.421,E2 -27382.421} C_VEL
LIN {X 0,Y 107.821,Z 753.262,A -85,B 0,C 180,E1 -27387.149,E2 -27387.149} C_VEL
LIN {X 0,Y 117.716,Z 755.77,A -85,B 0,C 180,E1 -27392.503,E2 -27392.503} C_VEL
LIN {X 0,Y 126.658,Z 756.826,A -85,B 0,C 180,E1 -27396.141,E2 -27396.141} C_VEL
LIN {X 0,Y 125.816,Z 756.984,A -85,B 0,C 180,E1 -27397.26,E2 -27397.26} C_VEL
LIN {X 0,Y 113.99,Z 756.748,A -85,B 0,C 180,E1 -27402.273,E2 -27402.273} C_VEL
LIN {X 0,Y 104.856,Z 755.406,A -85,B 0,C 180,E1 -27407.905,E2 -27407.905} C_VEL
LIN {X 0,Y 97.321,Z 752.996,A -85,B 0,C 180,E1 -27414.702,E2 -27414.702} C_VEL
LIN {X 0,Y 91.842,Z 749.402,A -85,B 0,C 180,E1 -27422.661,E2 -27422.661} C_VEL
LIN {X 0,Y 88.733,Z 744.547,A -85,B 0,C 180,E1 -27431.522,E2 -27431.522} C_VEL
LIN {X 0,Y 88.278,Z 738.258,A -85,B 0,C 180,E1 -27440.83,E2 -27440.83} C_VEL
LIN {X 0,Y 88.696,Z 734.343,A -85,B 0,C 180,E1 -27445.448,E2 -27445.448} C_VEL
LIN {X 0,Y 88.337,Z 729.109,A -85,B 0,C 180,E1 -27449.992,E2 -27449.992} C_VEL
LIN {X 0,Y 87.889,Z 722.892,A -85,B 0,C 180,E1 -27454.722,E2 -27454.722} C_VEL
LIN {X 0,Y 87.05,Z 719.088,A -85,B 0,C 180,E1 -27461.636,E2 -27461.636} C_VEL
LIN {X 0,Y 87.526,Z 714.07,A -85,B 0,C 180,E1 -27468.726,E2 -27468.726} C_VEL
LIN {X 0,Y 87.89,Z 712.609,A -85,B 0,C 180,E1 -27470.502,E2 -27470.502} C_VEL
LIN {X 0,Y 88.147,Z 709.687,A -85,B 0,C 180,E1 -27473.851,E2 -27473.851} C_VEL
LIN {X 0,Y 87.422,Z 704.353,A -85,B 0,C 180,E1 -27479.307,E2 -27479.307} C_VEL
LIN {X 0,Y 87.431,Z 698.374,A -85,B 0,C 180,E1 -27484.495,E2 -27484.495} C_VEL
LIN {X 0,Y 88.772,Z 694.443,A -85,B 0,C 180,E1 -27487.226,E2 -27487.226} C_VEL
LIN {X 0,Y 93.661,Z 684.706,A -85,B 0,C 180,E1 -27492.469,E2 -27492.469} C_VEL
LIN {X 0,Y 98.375,Z 674.839,A -85,B 0,C 180,E1 -27496.32,E2 -27496.32} C_VEL
LIN {X 0,Y 102.912,Z 664.027,A -85,B 0,C 180,E1 -27499.431,E2 -27499.431} C_VEL
LIN {X 0,Y 107.144,Z 651.911,A -85,B 0,C 180,E1 -27501.907,E2 -27501.907} C_VEL
LIN {X 0,Y 110.5,Z 639.198,A -85,B 0,C 180,E1 -27503.788,E2 -27503.788} C_VEL
LIN {X 0,Y 112.792,Z 626.674,A -85,B 0,C 180,E1 -27505.076,E2 -27505.076} C_VEL
LIN {X 0,Y 113.772,Z 617.953,A -85,B 0,C 180,E1 -27505.689,E2 -27505.689} C_VEL
LIN {X 0,Y 114.157,Z 571.768,A -85,B 0,C 180,E1 -27510.001,E2 -27510.001} C_VEL
LIN {X 0,Y 111.329,Z 562.326,A -85,B 0,C 180,E1 -27512.968,E2 -27512.968} C_VEL
LIN {X 0,Y 108.12,Z 553.344,A -85,B 0,C 180,E1 -27516.623,E2 -27516.623} C_VEL
LIN {X 0,Y 105.827,Z 547.751,A -85,B 0,C 180,E1 -27519.53,E2 -27519.53} C_VEL
LIN {X 0,Y 104.199,Z 544.027,A -85,B 0,C 180,E1 -27521.822,E2 -27521.822} C_VEL
LIN {X 0,Y 102.793,Z 541.731,A -85,B 0,C 180,E1 -27523.872,E2 -27523.872} C_VEL
LIN {X 0,Y 100.418,Z 538.148,A -85,B 0,C 180,E1 -27527.878,E2 -27527.878} C_VEL
LIN {X 0,Y 99.551,Z 536.965,A -85,B 0,C 180,E1 -27529.576,E2 -27529.576} C_VEL
LIN {X 0,Y 97.296,Z 533.44,A -85,B 0,C 180,E1 -27535.163,E2 -27535.163} C_VEL
LIN {X 0,Y 96.957,Z 532.597,A -85,B 0,C 180,E1 -27536.362,E2 -27536.362} C_VEL
LIN {X 0,Y 95.984,Z 531.789,A -85,B 0,C 180,E1 -27539.998,E2 -27539.998} C_VEL
LIN {X 0,Y 95.129,Z 531.614,A -85,B 0,C 180,E1 -27550.642,E2 -27550.642} C_VEL
LIN {X 0,Y 96.792,Z 532.881,A -85,B 0,C 180,E1 -27559.614,E2 -27559.614} C_VEL
LIN {X 0,Y 98.128,Z 535.864,A -85,B 0,C 180,E1 -27563.902,E2 -27563.902} C_VEL
LIN {X 0,Y 100.212,Z 538.122,A -85,B 0,C 180,E1 -27568.242,E2 -27568.242} C_VEL
LIN {X 0,Y 102.514,Z 541.618,A -85,B 0,C 180,E1 -27572.176,E2 -27572.176} C_VEL
LIN {X 0,Y 103.588,Z 543.13,A -85,B 0,C 180,E1 -27573.742,E2 -27573.742} C_VEL
LIN {X 0,Y 106.533,Z 547.688,A -85,B 0,C 180,E1 -27577.553,E2 -27577.553} C_VEL
LIN {X 0,Y 109.833,Z 553.103,A -85,B 0,C 180,E1 -27581.174,E2 -27581.174} C_VEL
LIN {X 0,Y 114.214,Z 561.548,A -85,B 0,C 180,E1 -27585.379,E2 -27585.379} C_VEL
LIN {X 0,Y 117.556,Z 569.288,A -85,B 0,C 180,E1 -27588.272,E2 -27588.272} C_VEL
LIN {X 0,Y 115.303,Z 601.694,A -85,B 0,C 180,E1 -27590.215,E2 -27590.215} C_VEL
LIN {X 0,Y 113.416,Z 615.268,A -85,B 0,C 180,E1 -27591.636,E2 -27591.636} C_VEL
LIN {X 0,Y 110.741,Z 627.61,A -85,B 0,C 180,E1 -27593.497,E2 -27593.497} C_VEL
LIN {X 0,Y 107.068,Z 640.035,A -85,B 0,C 180,E1 -27596.094,E2 -27596.094} C_VEL
LIN {X 0,Y 103.013,Z 651.149,A -85,B 0,C 180,E1 -27599.232,E2 -27599.232} C_VEL
LIN {X 0,Y 99.191,Z 660.166,A -85,B 0,C 180,E1 -27602.585,E2 -27602.585} C_VEL
LIN {X 0,Y 94.736,Z 669.464,A -85,B 0,C 180,E1 -27607.086,E2 -27607.086} C_VEL
LIN {X 0,Y 90.115,Z 678.477,A -85,B 0,C 180,E1 -27613.003,E2 -27613.003} C_VEL
LIN {X 0,Y 86.219,Z 685.764,A -85,B 0,C 180,E1 -27619.398,E2 -27619.398} C_VEL
LIN {X 0,Y 83.739,Z 690.756,A -85,B 0,C 180,E1 -27625.194,E2 -27625.194} C_VEL
LIN {X 0,Y 81.627,Z 695.624,A -85,B 0,C 180,E1 -27632.476,E2 -27632.476} C_VEL
LIN {X 0,Y 80.743,Z 699.371,A -85,B 0,C 180,E1 -27640.034,E2 -27640.034} C_VEL
LIN {X 0,Y 81.029,Z 702.031,A -85,B 0,C 180,E1 -27647.437,E2 -27647.437} C_VEL
LIN {X 0,Y 82.596,Z 703.886,A -85,B 0,C 180,E1 -27655.187,E2 -27655.187} C_VEL
LIN {X 0,Y 84.312,Z 704.578,A -85,B 0,C 180,E1 -27660.018,E2 -27660.018} C_VEL
LIN {X 0,Y 87.839,Z 704.808,A -85,B 0,C 180,E1 -27666.864,E2 -27666.864} C_VEL
LIN {X 0,Y 92.441,Z 704.108,A -85,B 0,C 180,E1 -27673.186,E2 -27673.186} C_VEL
LIN {X 0,Y 81.63,Z 705.853,A -85,B 0,C 180,E1 -27688.899,E2 -27688.899} C_VEL
LIN {X 0,Y 79.436,Z 706.413,A -85,B 0,C 180,E1 -27699.446,E2 -27699.446} C_VEL
LIN {X 0,Y 79.461,Z 707.572,A -85,B 0,C 180,E1 -27700.632,E2 -27700.632} C_VEL
LIN {X 0,Y 79.06,Z 717.6,A -85,B 0,C 180,E1 -27707.955,E2 -27707.955} C_VEL
LIN {X 0,Y 79.373,Z 725.463,A -85,B 0,C 180,E1 -27714.922,E2 -27714.922} C_VEL
LIN {X 0,Y 81.15,Z 733.704,A -85,B 0,C 180,E1 -27723.726,E2 -27723.726} C_VEL
LIN {X 0,Y 84.654,Z 740.385,A -85,B 0,C 180,E1 -27731.981,E2 -27731.981} C_VEL
LIN {X 0,Y 90.886,Z 746.525,A -85,B 0,C 180,E1 -27740.365,E2 -27740.365} C_VEL
LIN {X 0,Y 99.105,Z 751.304,A -85,B 0,C 180,E1 -27747.45,E2 -27747.45} C_VEL
LIN {X 0,Y 109.749,Z 754.881,A -85,B 0,C 180,E1 -27753.635,E2 -27753.635} C_VEL
LIN {X 0,Y 115.26,Z 756.077,A -85,B 0,C 180,E1 -27756.083,E2 -27756.083} C_VEL
LIN {X 0,Y 114.758,Z 756.188,A -85,B 0,C 180,E1 -27757.227,E2 -27757.227} C_VEL
LIN {X 0,Y 103.38,Z 754.761,A -85,B 0,C 180,E1 -27762.832,E2 -27762.832} C_VEL
LIN {X 0,Y 95.589,Z 752.687,A -85,B 0,C 180,E1 -27768.561,E2 -27768.561} C_VEL
LIN {X 0,Y 88.536,Z 749.336,A -85,B 0,C 180,E1 -27776.235,E2 -27776.235} C_VEL
LIN {X 0,Y 83.848,Z 744.782,A -85,B 0,C 180,E1 -27785.214,E2 -27785.214} C_VEL
LIN {X 0,Y 81.861,Z 738.92,A -85,B 0,C 180,E1 -27795.066,E2 -27795.066} C_VEL
LIN {X 0,Y 82.112,Z 733.401,A -85,B 0,C 180,E1 -27802.615,E2 -27802.615} C_VEL
LIN {X 0,Y 82.075,Z 729.883,A -85,B 0,C 180,E1 -27806.31,E2 -27806.31} C_VEL
LIN {X 0,Y 81.4,Z 722.908,A -85,B 0,C 180,E1 -27812.156,E2 -27812.156} C_VEL
LIN {X 0,Y 80.095,Z 719.205,A -85,B 0,C 180,E1 -27820.099,E2 -27820.099} C_VEL
LIN {X 0,Y 80.283,Z 714.49,A -85,B 0,C 180,E1 -27827.833,E2 -27827.833} C_VEL
LIN {X 0,Y 82.116,Z 708.588,A -85,B 0,C 180,E1 -27835.327,E2 -27835.327} C_VEL
LIN {X 0,Y 85.374,Z 701.205,A -85,B 0,C 180,E1 -27842.34,E2 -27842.34} C_VEL
LIN {X 0,Y 88.772,Z 694.443,A -85,B 0,C 180,E1 -27847.226,E2 -27847.226} C_VEL
LIN {X 0,Y 90.281,Z 690.382,A -85,B 0,C 180,E1 -27849.8,E2 -27849.8} C_VEL
LIN {X 0,Y 91.355,Z 683.337,A -85,B 0,C 180,E1 -27854.17,E2 -27854.17} C_VEL
LIN {X 0,Y 92.65,Z 675.875,A -85,B 0,C 180,E1 -27858.165,E2 -27858.165} C_VEL
LIN {X 0,Y 94.355,Z 671.071,A -85,B 0,C 180,E1 -27859.999,E2 -27859.999} C_VEL
LIN {X 0,Y 99.034,Z 659.943,A -85,B 0,C 180,E1 -27862.962,E2 -27862.962} C_VEL
LIN {X 0,Y 103.173,Z 647.984,A -85,B 0,C 180,E1 -27865.241,E2 -27865.241} C_VEL
LIN {X 0,Y 106.382,Z 635.461,A -85,B 0,C 180,E1 -27866.936,E2 -27866.936} C_VEL
LIN {X 0,Y 108.664,Z 622.588,A -85,B 0,C 180,E1 -27868.087,E2 -27868.087} C_VEL
LIN {X 0,Y 109.138,Z 616.227,A -85,B 0,C 180,E1 -27868.649,E2 -27868.649} C_VEL
LIN {X 0,Y 109.872,Z 574.153,A -85,B 0,C 180,E1 -27872.716,E2 -27872.716} C_VEL
LIN {X 0,Y 107.187,Z 564.776,A -85,B 0,C 180,E1 -27875.982,E2 -27875.982} C_VEL
LIN {X 0,Y 104.699,Z 557.335,A -85,B 0,C 180,E1 -27879.299,E2 -27879.299} C_VEL
LIN {X 0,Y 102.063,Z 550.275,A -85,B 0,C 180,E1 -27883.328,E2 -27883.328} C_VEL
LIN {X 0,Y 100.652,Z 547.874,A -85,B 0,C 180,E1 -27885.607,E2 -27885.607} C_VEL
LIN {X 0,Y 98.128,Z 543.707,A -85,B 0,C 180,E1 -27890.536,E2 -27890.536} C_VEL
LIN {X 0,Y 95.939,Z 539.986,A -85,B 0,C 180,E1 -27896.586,E2 -27896.586} C_VEL
LIN {X 0,Y 95.598,Z 539.364,A -85,B 0,C 180,E1 -27897.892,E2 -27897.892} C_VEL
LIN {X 0,Y 94.677,Z 538.698,A -85,B 0,C 180,E1 -27902.126,E2 -27902.126} C_VEL
LIN {X 0,Y 94.255,Z 538.68,A -85,B 0,C 180,E1 -27910.742,E2 -27910.742} C_VEL
LIN {X 0,Y 95.611,Z 539.903,A -85,B 0,C 180,E1 -27918.693,E2 -27918.693} C_VEL
LIN {X 0,Y 97.274,Z 543.282,A -85,B 0,C 180,E1 -27924.125,E2 -27924.125} C_VEL
LIN {X 0,Y 98.605,Z 544.821,A -85,B 0,C 180,E1 -27927.041,E2 -27927.041} C_VEL
LIN {X 0,Y 101.517,Z 549.413,A -85,B 0,C 180,E1 -27932.258,E2 -27932.258} C_VEL
LIN {X 0,Y 104.491,Z 554.297,A -85,B 0,C 180,E1 -27936.448,E2 -27936.448} C_VEL
LIN {X 0,Y 107.941,Z 560.619,A -85,B 0,C 180,E1 -27940.523,E2 -27940.523} C_VEL
LIN {X 0,Y 111.355,Z 567.967,A -85,B 0,C 180,E1 -27944.062,E2 -27944.062} C_VEL
LIN {X 0,Y 112.967,Z 571.817,A -85,B 0,C 180,E1 -27945.614,E2 -27945.614} C_VEL
LIN {X 0,Y 110.647,Z 602.809,A -85,B 0,C 180,E1 -27947.519,E2 -27947.519} C_VEL
LIN {X 0,Y 108.646,Z 616.421,A -85,B 0,C 180,E1 -27948.985,E2 -27948.985} C_VEL
LIN {X 0,Y 105.774,Z 628.774,A -85,B 0,C 180,E1 -27950.869,E2 -27950.869} C_VEL
LIN {X 0,Y 101.876,Z 641.162,A -85,B 0,C 180,E1 -27953.496,E2 -27953.496} C_VEL
LIN {X 0,Y 97.552,Z 652.255,A -85,B 0,C 180,E1 -27956.687,E2 -27956.687} C_VEL
LIN {X 0,Y 92.989,Z 662.254,A -85,B 0,C 180,E1 -27960.585,E2 -27960.585} C_VEL
LIN {X 0,Y 88.277,Z 671.334,A -85,B 0,C 180,E1 -27965.302,E2 -27965.302} C_VEL
LIN {X 0,Y 83.365,Z 680.206,A -85,B 0,C 180,E1 -27971.579,E2 -27971.579} C_VEL
LIN {X 0,Y 79.111,Z 687.588,A -85,B 0,C 180,E1 -27978.748,E2 -27978.748} C_VEL
LIN {X 0,Y 75.763,Z 693.947,A -85,B 0,C 180,E1 -27987.351,E2 -27987.351} C_VEL
LIN {X 0,Y 74.068,Z 698.323,A -85,B 0,C 180,E1 -27995.454,E2 -27995.454} C_VEL
LIN {X 0,Y 73.673,Z 700.669,A -85,B 0,C 180,E1 -28001.008,E2 -28001.008} C_VEL
LIN {X 0,Y 74.099,Z 703.061,A -85,B 0,C 180,E1 -28008.482,E2 -28008.482} C_VEL
LIN {X 0,Y 76.117,Z 705.007,A -85,B 0,C 180,E1 -28017.504,E2 -28017.504} C_VEL
LIN {X 0,Y 78.114,Z 705.632,A -85,B 0,C 180,E1 -28022.682,E2 -28022.682} C_VEL
LIN {X 0,Y 83.749,Z 705.613,A -85,B 0,C 180,E1 -28032.181,E2 -28032.181} C_VEL
LIN {X 0,Y 81.412,Z 706.079,A -85,B 0,C 180,E1 -28036.324,E2 -28036.324} C_VEL
LIN {X 0,Y 73.74,Z 707.725,A -85,B 0,C 180,E1 -28051.543,E2 -28051.543} C_VEL
LIN {X 0,Y 72.48,Z 708.529,A -85,B 0,C 180,E1 -28063.277,E2 -28063.277} C_VEL
LIN {X 0,Y 72.503,Z 718.835,A -85,B 0,C 180,E1 -28071.905,E2 -28071.905} C_VEL
LIN {X 0,Y 73.419,Z 726.84,A -85,B 0,C 180,E1 -28080.002,E2 -28080.002} C_VEL
LIN {X 0,Y 76.149,Z 734.778,A -85,B 0,C 180,E1 -28089.297,E2 -28089.297} C_VEL
LIN {X 0,Y 81.746,Z 742.181,A -85,B 0,C 180,E1 -28098.942,E2 -28098.942} C_VEL
LIN {X 0,Y 88.356,Z 747.33,A -85,B 0,C 180,E1 -28105.945,E2 -28105.945} C_VEL
LIN {X 0,Y 97.729,Z 751.974,A -85,B 0,C 180,E1 -28112.641,E2 -28112.641} C_VEL
LIN {X 0,Y 105.089,Z 754.46,A -85,B 0,C 180,E1 -28116.618,E2 -28116.618} C_VEL
LIN {X 0,Y 95.007,Z 752.311,A -85,B 0,C 180,E1 -28122.281,E2 -28122.281} C_VEL
LIN {X 0,Y 86.517,Z 749.139,A -85,B 0,C 180,E1 -28129.459,E2 -28129.459} C_VEL
LIN {X 0,Y 80.119,Z 744.86,A -85,B 0,C 180,E1 -28138.234,E2 -28138.234} C_VEL
LIN {X 0,Y 76.351,Z 739.289,A -85,B 0,C 180,E1 -28148.386,E2 -28148.386} C_VEL
LIN {X 0,Y 75.512,Z 734.221,A -85,B 0,C 180,E1 -28156.536,E2 -28156.536} C_VEL
LIN {X 0,Y 75.837,Z 729.019,A -85,B 0,C 180,E1 -28163.339,E2 -28163.339} C_VEL
LIN {X 0,Y 75.017,Z 722.773,A -85,B 0,C 180,E1 -28169.32,E2 -28169.32} C_VEL
LIN {X 0,Y 73.173,Z 719.233,A -85,B 0,C 180,E1 -28178.274,E2 -28178.274} C_VEL
LIN {X 0,Y 73.069,Z 714.82,A -85,B 0,C 180,E1 -28186.761,E2 -28186.761} C_VEL
LIN {X 0,Y 75.177,Z 708.169,A -85,B 0,C 180,E1 -28196.353,E2 -28196.353} C_VEL
LIN {X 0,Y 78.661,Z 700.962,A -85,B 0,C 180,E1 -28203.935,E2 -28203.935} C_VEL
LIN {X 0,Y 83.179,Z 692.658,A -85,B 0,C 180,E1 -28210.239,E2 -28210.239} C_VEL
LIN {X 0,Y 88.529,Z 682.797,A -85,B 0,C 180,E1 -28215.589,E2 -28215.589} C_VEL
LIN {X 0,Y 93.584,Z 672.734,A -85,B 0,C 180,E1 -28219.485,E2 -28219.485} C_VEL
LIN {X 0,Y 94.355,Z 671.071,A -85,B 0,C 180,E1 -28219.999,E2 -28219.999} C_VEL
LIN {X 0,Y 96.012,Z 666.176,A -85,B 0,C 180,E1 -28221.681,E2 -28221.681} C_VEL
LIN {X 0,Y 97.225,Z 657.861,A -85,B 0,C 180,E1 -28224.852,E2 -28224.852} C_VEL
LIN {X 0,Y 98.275,Z 649.255,A -85,B 0,C 180,E1 -28227.698,E2 -28227.698} C_VEL
LIN {X 0,Y 99.563,Z 643.78,A -85,B 0,C 180,E1 -28228.813,E2 -28228.813} C_VEL
LIN {X 0,Y 102.754,Z 630.804,A -85,B 0,C 180,E1 -28230.408,E2 -28230.408} C_VEL
LIN {X 0,Y 104.602,Z 619.586,A -85,B 0,C 180,E1 -28231.319,E2 -28231.319} C_VEL
LIN {X 0,Y 105.864,Z 576.687,A -85,B 0,C 180,E1 -28235.615,E2 -28235.615} C_VEL
LIN {X 0,Y 103.517,Z 567.843,A -85,B 0,C 180,E1 -28238.987,E2 -28238.987} C_VEL
LIN {X 0,Y 101.21,Z 560.216,A -85,B 0,C 180,E1 -28242.704,E2 -28242.704} C_VEL
LIN {X 0,Y 99.415,Z 555.292,A -85,B 0,C 180,E1 -28245.947,E2 -28245.947} C_VEL
LIN {X 0,Y 96.523,Z 550.179,A -85,B 0,C 180,E1 -28252.016,E2 -28252.016} C_VEL
LIN {X 0,Y 94.57,Z 546.313,A -85,B 0,C 180,E1 -28258.401,E2 -28258.401} C_VEL
LIN {X 0,Y 93.501,Z 545.629,A -85,B 0,C 180,E1 -28264.309,E2 -28264.309} C_VEL
LIN {X 0,Y 93.51,Z 545.888,A -85,B 0,C 180,E1 -28272.334,E2 -28272.334} C_VEL
LIN {X 0,Y 94.437,Z 546.73,A -85,B 0,C 180,E1 -28277.595,E2 -28277.595} C_VEL
LIN {X 0,Y 96.123,Z 550.304,A -85,B 0,C 180,E1 -28283.598,E2 -28283.598} C_VEL
LIN {X 0,Y 97.078,Z 551.579,A -85,B 0,C 180,E1 -28285.88,E2 -28285.88} C_VEL
LIN {X 0,Y 99.559,Z 555.776,A -85,B 0,C 180,E1 -28290.787,E2 -28290.787} C_VEL
LIN {X 0,Y 102.114,Z 560.261,A -85,B 0,C 180,E1 -28294.777,E2 -28294.777} C_VEL
LIN {X 0,Y 105.169,Z 566.321,A -85,B 0,C 180,E1 -28298.796,E2 -28298.796} C_VEL
LIN {X 0,Y 108.058,Z 573.067,A -85,B 0,C 180,E1 -28302.138,E2 -28302.138} C_VEL
LIN {X 0,Y 108.62,Z 574.549,A -85,B 0,C 180,E1 -28302.754,E2 -28302.754} C_VEL
LIN {X 0,Y 106.307,Z 603.664,A -85,B 0,C 180,E1 -28304.585,E2 -28304.585} C_VEL
LIN {X 0,Y 104.257,Z 616.824,A -85,B 0,C 180,E1 -28305.989,E2 -28305.989} C_VEL
LIN {X 0,Y 101.349,Z 628.932,A -85,B 0,C 180,E1 -28307.805,E2 -28307.805} C_VEL
LIN {X 0,Y 97.506,Z 640.72,A -85,B 0,C 180,E1 -28310.241,E2 -28310.241} C_VEL
LIN {X 0,Y 92.902,Z 652.064,A -85,B 0,C 180,E1 -28313.444,E2 -28313.444} C_VEL
LIN {X 0,Y 87.967,Z 662.329,A -85,B 0,C 180,E1 -28317.375,E2 -28317.375} C_VEL
LIN {X 0,Y 82.859,Z 671.58,A -85,B 0,C 180,E1 -28322.202,E2 -28322.202} C_VEL
LIN {X 0,Y 77.502,Z 680.568,A -85,B 0,C 180,E1 -28328.742,E2 -28328.742} C_VEL
LIN {X 0,Y 73.28,Z 687.262,A -85,B 0,C 180,E1 -28335.366,E2 -28335.366} C_VEL
LIN {X 0,Y 69.505,Z 693.725,A -85,B 0,C 180,E1 -28344.206,E2 -28344.206} C_VEL
LIN {X 0,Y 67.335,Z 698.37,A -85,B 0,C 180,E1 -28353.001,E2 -28353.001} C_VEL
LIN {X 0,Y 66.63,Z 701.934,A -85,B 0,C 180,E1 -28362.189,E2 -28362.189} C_VEL
LIN {X 0,Y 67.19,Z 704.085,A -85,B 0,C 180,E1 -28369.721,E2 -28369.721} C_VEL
LIN {X 0,Y 69.779,Z 706.12,A -85,B 0,C 180,E1 -28380.249,E2 -28380.249} C_VEL
LIN {X 0,Y 72.114,Z 706.666,A -85,B 0,C 180,E1 -28385.796,E2 -28385.796} C_VEL
LIN {X 0,Y 75.869,Z 706.802,A -85,B 0,C 180,E1 -28392.181,E2 -28392.181} C_VEL
LIN {X 0,Y 72.639,Z 707.538,A -85,B 0,C 180,E1 -28397.372,E2 -28397.372} C_VEL
LIN {X 0,Y 65.982,Z 709.471,A -85,B 0,C 180,E1 -28414.785,E2 -28414.785} C_VEL
LIN {X 0,Y 65.678,Z 710.409,A -85,B 0,C 180,E1 -28427.36,E2 -28427.36} C_VEL
LIN {X 0,Y 65.827,Z 712.067,A -85,B 0,C 180,E1 -28429.234,E2 -28429.234} C_VEL
LIN {X 0,Y 66.342,Z 720.081,A -85,B 0,C 180,E1 -28436.966,E2 -28436.966} C_VEL
LIN {X 0,Y 68.517,Z 729.248,A -85,B 0,C 180,E1 -28447.369,E2 -28447.369} C_VEL
LIN {X 0,Y 73.756,Z 737.964,A -85,B 0,C 180,E1 -28458.541,E2 -28458.541} C_VEL
LIN {X 0,Y 79.908,Z 743.694,A -85,B 0,C 180,E1 -28466.09,E2 -28466.09} C_VEL
LIN {X 0,Y 89.175,Z 749.247,A -85,B 0,C 180,E1 -28473.484,E2 -28473.484} C_VEL
LIN {X 0,Y 94.446,Z 751.574,A -85,B 0,C 180,E1 -28476.536,E2 -28476.536} C_VEL
LIN {X 0,Y 85.801,Z 748.857,A -85,B 0,C 180,E1 -28482.496,E2 -28482.496} C_VEL
LIN {X 0,Y 77.711,Z 744.758,A -85,B 0,C 180,E1 -28490.713,E2 -28490.713} C_VEL
LIN {X 0,Y 71.656,Z 738.908,A -85,B 0,C 180,E1 -28501.977,E2 -28501.977} C_VEL
LIN {X 0,Y 69.545,Z 732.911,A -85,B 0,C 180,E1 -28512.342,E2 -28512.342} C_VEL
LIN {X 0,Y 69.563,Z 726.792,A -85,B 0,C 180,E1 -28521.274,E2 -28521.274} C_VEL
LIN {X 0,Y 68.956,Z 722.651,A -85,B 0,C 180,E1 -28525.606,E2 -28525.606} C_VEL
LIN {X 0,Y 66.318,Z 719.166,A -85,B 0,C 180,E1 -28536.073,E2 -28536.073} C_VEL
LIN {X 0,Y 65.961,Z 714.555,A -85,B 0,C 180,E1 -28546.469,E2 -28546.469} C_VEL
LIN {X 0,Y 67.759,Z 708.776,A -85,B 0,C 180,E1 -28556.144,E2 -28556.144} C_VEL
LIN {X 0,Y 71.287,Z 701.927,A -85,B 0,C 180,E1 -28564.521,E2 -28564.521} C_VEL
LIN {X 0,Y 76.327,Z 693.442,A -85,B 0,C 180,E1 -28571.899,E2 -28571.899} C_VEL
LIN {X 0,Y 81.404,Z 684.831,A -85,B 0,C 180,E1 -28577.197,E2 -28577.197} C_VEL
LIN {X 0,Y 87.252,Z 674.201,A -85,B 0,C 180,E1 -28581.74,E2 -28581.74} C_VEL
LIN {X 0,Y 92.27,Z 663.663,A -85,B 0,C 180,E1 -28584.952,E2 -28584.952} C_VEL
LIN {X 0,Y 96.909,Z 652.114,A -85,B 0,C 180,E1 -28587.452,E2 -28587.452} C_VEL
LIN {X 0,Y 99.563,Z 643.78,A -85,B 0,C 180,E1 -28588.813,E2 -28588.813} C_VEL
LIN {X 0,Y 100.705,Z 638.257,A -85,B 0,C 180,E1 -28589.818,E2 -28589.818} C_VEL
LIN {X 0,Y 100.993,Z 629.184,A -85,B 0,C 180,E1 -28592.087,E2 -28592.087} C_VEL
LIN {X 0,Y 100.731,Z 621.837,A -85,B 0,C 180,E1 -28593.907,E2 -28593.907} C_VEL
LIN {X 0,Y 100.824,Z 614.181,A -85,B 0,C 180,E1 -28595.155,E2 -28595.155} C_VEL
LIN {X 0,Y 102.095,Z 579.056,A -85,B 0,C 180,E1 -28598.812,E2 -28598.812} C_VEL
LIN {X 0,Y 100.124,Z 570.852,A -85,B 0,C 180,E1 -28602.246,E2 -28602.246} C_VEL
LIN {X 0,Y 98.141,Z 563.73,A -85,B 0,C 180,E1 -28606.155,E2 -28606.155} C_VEL
LIN {X 0,Y 97.22,Z 560.918,A -85,B 0,C 180,E1 -28608.175,E2 -28608.175} C_VEL
LIN {X 0,Y 95.003,Z 556.711,A -85,B 0,C 180,E1 -28613.485,E2 -28613.485} C_VEL
LIN {X 0,Y 93.303,Z 553.087,A -85,B 0,C 180,E1 -28619.998,E2 -28619.998} C_VEL
LIN {X 0,Y 92.422,Z 552.652,A -85,B 0,C 180,E1 -28628.746,E2 -28628.746} C_VEL
LIN {X 0,Y 93.301,Z 553.629,A -85,B 0,C 180,E1 -28636.565,E2 -28636.565} C_VEL
LIN {X 0,Y 95.056,Z 557.383,A -85,B 0,C 180,E1 -28643.251,E2 -28643.251} C_VEL
LIN {X 0,Y 96.233,Z 559.607,A -85,B 0,C 180,E1 -28646.262,E2 -28646.262} C_VEL
LIN {X 0,Y 97.662,Z 562.115,A -85,B 0,C 180,E1 -28649.242,E2 -28649.242} C_VEL
LIN {X 0,Y 100.023,Z 566.612,A -85,B 0,C 180,E1 -28653.338,E2 -28653.338} C_VEL
LIN {X 0,Y 103.007,Z 573.355,A -85,B 0,C 180,E1 -28657.686,E2 -28657.686} C_VEL
LIN {X 0,Y 104.549,Z 577.325,A -85,B 0,C 180,E1 -28659.692,E2 -28659.692} C_VEL
LIN {X 0,Y 102.204,Z 604.703,A -85,B 0,C 180,E1 -28661.435,E2 -28661.435} C_VEL
LIN {X 0,Y 99.952,Z 618.137,A -85,B 0,C 180,E1 -28662.864,E2 -28662.864} C_VEL
LIN {X 0,Y 96.606,Z 631.009,A -85,B 0,C 180,E1 -28664.832,E2 -28664.832} C_VEL
LIN {X 0,Y 92.201,Z 643.358,A -85,B 0,C 180,E1 -28667.44,E2 -28667.44} C_VEL
LIN {X 0,Y 87.323,Z 654.406,A -85,B 0,C 180,E1 -28670.679,E2 -28670.679} C_VEL
LIN {X 0,Y 82.113,Z 664.362,A -85,B 0,C 180,E1 -28674.72,E2 -28674.72} C_VEL
LIN {X 0,Y 76.689,Z 673.418,A -85,B 0,C 180,E1 -28679.743,E2 -28679.743} C_VEL
LIN {X 0,Y 70.895,Z 682.283,A -85,B 0,C 180,E1 -28686.649,E2 -28686.649} C_VEL
LIN {X 0,Y 66.543,Z 688.662,A -85,B 0,C 180,E1 -28693.594,E2 -28693.594} C_VEL
LIN {X 0,Y 62.383,Z 695.152,A -85,B 0,C 180,E1 -28703.542,E2 -28703.542} C_VEL
LIN {X 0,Y 60.172,Z 699.698,A -85,B 0,C 180,E1 -28713.359,E2 -28713.359} C_VEL
LIN {X 0,Y 59.608,Z 703.175,A -85,B 0,C 180,E1 -28723.651,E2 -28723.651} C_VEL
LIN {X 0,Y 60.295,Z 705.087,A -85,B 0,C 180,E1 -28731.182,E2 -28731.182} C_VEL
LIN {X 0,Y 63.628,Z 707.201,A -85,B 0,C 180,E1 -28743.536,E2 -28743.536} C_VEL
LIN {X 0,Y 66.365,Z 707.701,A -85,B 0,C 180,E1 -28749.462,E2 -28749.462} C_VEL
LIN {X 0,Y 67.32,Z 707.968,A -85,B 0,C 180,E1 -28753.052,E2 -28753.052} C_VEL
LIN {X 0,Y 58.536,Z 711.035,A -85,B 0,C 180,E1 -28778.891,E2 -28778.891} C_VEL
LIN {X 0,Y 59.451,Z 712.314,A -85,B 0,C 180,E1 -28793.213,E2 -28793.213} C_VEL
LIN {X 0,Y 60.75,Z 721.427,A -85,B 0,C 180,E1 -28803.318,E2 -28803.318} C_VEL
LIN {X 0,Y 64.177,Z 730.18,A -85,B 0,C 180,E1 -28814.267,E2 -28814.267} C_VEL
LIN {X 0,Y 69.708,Z 737.479,A -85,B 0,C 180,E1 -28823.786,E2 -28823.786} C_VEL
LIN {X 0,Y 78.357,Z 744.354,A -85,B 0,C 180,E1 -28832.56,E2 -28832.56} C_VEL
LIN {X 0,Y 83.351,Z 747.278,A -85,B 0,C 180,E1 -28836.175,E2 -28836.175} C_VEL
LIN {X 0,Y 81.387,Z 746.662,A -85,B 0,C 180,E1 -28838.985,E2 -28838.985} C_VEL
LIN {X 0,Y 72.717,Z 742.219,A -85,B 0,C 180,E1 -28847.414,E2 -28847.414} C_VEL
LIN {X 0,Y 66.542,Z 736.574,A -85,B 0,C 180,E1 -28858.112,E2 -28858.112} C_VEL
LIN {X 0,Y 63.593,Z 729.623,A -85,B 0,C 180,E1 -28870.626,E2 -28870.626} C_VEL
LIN {X 0,Y 63.425,Z 724.343,A -85,B 0,C 180,E1 -28878.808,E2 -28878.808} C_VEL
LIN {X 0,Y 63.034,Z 722.287,A -85,B 0,C 180,E1 -28881.574,E2 -28881.574} C_VEL
LIN {X 0,Y 59.618,Z 719.05,A -85,B 0,C 180,E1 -28893.368,E2 -28893.368} C_VEL
LIN {X 0,Y 58.782,Z 715.215,A -85,B 0,C 180,E1 -28903.823,E2 -28903.823} C_VEL
LIN {X 0,Y 59.995,Z 710.237,A -85,B 0,C 180,E1 -28914.192,E2 -28914.192} C_VEL
LIN {X 0,Y 63.21,Z 703.992,A -85,B 0,C 180,E1 -28923.761,E2 -28923.761} C_VEL
LIN {X 0,Y 68.116,Z 696.261,A -85,B 0,C 180,E1 -28932.103,E2 -28932.103} C_VEL
LIN {X 0,Y 73.468,Z 688.091,A -85,B 0,C 180,E1 -28938.22,E2 -28938.22} C_VEL
LIN {X 0,Y 79.837,Z 677.808,A -85,B 0,C 180,E1 -28943.428,E2 -28943.428} C_VEL
LIN {X 0,Y 85.671,Z 666.992,A -85,B 0,C 180,E1 -28947.215,E2 -28947.215} C_VEL
LIN {X 0,Y 90.441,Z 656.533,A -85,B 0,C 180,E1 -28949.81,E2 -28949.81} C_VEL
LIN {X 0,Y 94.993,Z 643.975,A -85,B 0,C 180,E1 -28952.013,E2 -28952.013} C_VEL
LIN {X 0,Y 98.549,Z 630.524,A -85,B 0,C 180,E1 -28953.655,E2 -28953.655} C_VEL
LIN {X 0,Y 100.461,Z 619.736,A -85,B 0,C 180,E1 -28954.548,E2 -28954.548} C_VEL
LIN {X 0,Y 100.824,Z 614.181,A -85,B 0,C 180,E1 -28955.155,E2 -28955.155} C_VEL
LIN {X 0,Y 100.775,Z 608.487,A -85,B 0,C 180,E1 -28956.053,E2 -28956.053} C_VEL
LIN {X 0,Y 98.578,Z 590.591,A -85,B 0,C 180,E1 -28960.868,E2 -28960.868} C_VEL
LIN {X 0,Y 98.585,Z 584.884,A -85,B 0,C 180,E1 -28961.765,E2 -28961.765} C_VEL
LIN {X 0,Y 98.656,Z 581.513,A -85,B 0,C 180,E1 -28962.241,E2 -28962.241} C_VEL
LIN {X 0,Y 96.854,Z 572.948,A -85,B 0,C 180,E1 -28966.233,E2 -28966.233} C_VEL
LIN {X 0,Y 95.459,Z 567.269,A -85,B 0,C 180,E1 -28969.774,E2 -28969.774} C_VEL
LIN {X 0,Y 93.493,Z 563.127,A -85,B 0,C 180,E1 -28975.183,E2 -28975.183} C_VEL
LIN {X 0,Y 92.203,Z 559.965,A -85,B 0,C 180,E1 -28981.09,E2 -28981.09} C_VEL
LIN {X 0,Y 91.544,Z 559.709,A -85,B 0,C 180,E1 -28988.831,E2 -28988.831} C_VEL
LIN {X 0,Y 92.239,Z 560.658,A -85,B 0,C 180,E1 -28995.785,E2 -28995.785} C_VEL
LIN {X 0,Y 94.122,Z 564.924,A -85,B 0,C 180,E1 -29003.337,E2 -29003.337} C_VEL
LIN {X 0,Y 95.958,Z 568.683,A -85,B 0,C 180,E1 -29007.892,E2 -29007.892} C_VEL
LIN {X 0,Y 98.053,Z 573.209,A -85,B 0,C 180,E1 -29011.958,E2 -29011.958} C_VEL
LIN {X 0,Y 100.477,Z 579.361,A -85,B 0,C 180,E1 -29015.928,E2 -29015.928} C_VEL
LIN {X 0,Y 100.808,Z 580.255,A -85,B 0,C 180,E1 -29016.425,E2 -29016.425} C_VEL
LIN {X 0,Y 98.379,Z 606.206,A -85,B 0,C 180,E1 -29018.083,E2 -29018.083} C_VEL
LIN {X 0,Y 95.909,Z 619.663,A -85,B 0,C 180,E1 -29019.48,E2 -29019.48} C_VEL
LIN {X 0,Y 92.471,Z 632.081,A -85,B 0,C 180,E1 -29021.376,E2 -29021.376} C_VEL
LIN {X 0,Y 87.806,Z 644.413,A -85,B 0,C 180,E1 -29023.927,E2 -29023.927} C_VEL
LIN {X 0,Y 82.66,Z 655.432,A -85,B 0,C 180,E1 -29027.154,E2 -29027.154} C_VEL
LIN {X 0,Y 77.668,Z 664.397,A -85,B 0,C 180,E1 -29030.709,E2 -29030.709} C_VEL
LIN {X 0,Y 71.777,Z 673.623,A -85,B 0,C 180,E1 -29035.748,E2 -29035.748} C_VEL
LIN {X 0,Y 65.436,Z 682.608,A -85,B 0,C 180,E1 -29042.853,E2 -29042.853} C_VEL
LIN {X 0,Y 59.897,Z 690.03,A -85,B 0,C 180,E1 -29051.398,E2 -29051.398} C_VEL
LIN {X 0,Y 56.45,Z 694.835,A -85,B 0,C 180,E1 -29059.249,E2 -29059.249} C_VEL
LIN {X 0,Y 53.56,Z 699.681,A -85,B 0,C 180,E1 -29070.013,E2 -29070.013} C_VEL
LIN {X 0,Y 52.535,Z 703.415,A -85,B 0,C 180,E1 -29081.589,E2 -29081.589} C_VEL
LIN {X 0,Y 53.483,Z 706.134,A -85,B 0,C 180,E1 -29093.231,E2 -29093.231} C_VEL
LIN {X 0,Y 55.197,Z 707.432,A -85,B 0,C 180,E1 -29100.631,E2 -29100.631} C_VEL
LIN {X 0,Y 58.907,Z 708.523,A -85,B 0,C 180,E1 -29110.085,E2 -29110.085} C_VEL
LIN {X 0,Y 59.367,Z 708.779,A -85,B 0,C 180,E1 -29112.718,E2 -29112.718} C_VEL
LIN {X 0,Y 51.381,Z 712.487,A -85,B 0,C 180,E1 -29144.126,E2 -29144.126} C_VEL
LIN {X 0,Y 53.622,Z 714.005,A -85,B 0,C 180,E1 -29160.003,E2 -29160.003} C_VEL
LIN {X 0,Y 57.178,Z 725.137,A -85,B 0,C 180,E1 -29174.233,E2 -29174.233} C_VEL
LIN {X 0,Y 61.619,Z 732.003,A -85,B 0,C 180,E1 -29183.347,E2 -29183.347} C_VEL
LIN {X 0,Y 70.157,Z 739.959,A -85,B 0,C 180,E1 -29193.436,E2 -29193.436} C_VEL
LIN {X 0,Y 73.904,Z 742.573,A -85,B 0,C 180,E1 -29196.481,E2 -29196.481} C_VEL
LIN {X 0,Y 72.47,Z 741.993,A -85,B 0,C 180,E1 -29199.106,E2 -29199.106} C_VEL
LIN {X 0,Y 64.278,Z 736.635,A -85,B 0,C 180,E1 -29208.989,E2 -29208.989} C_VEL
LIN {X 0,Y 59.013,Z 729.939,A -85,B 0,C 180,E1 -29221.539,E2 -29221.539} C_VEL
LIN {X 0,Y 57.484,Z 722.916,A -85,B 0,C 180,E1 -29234.021,E2 -29234.021} C_VEL
LIN {X 0,Y 57.404,Z 721.884,A -85,B 0,C 180,E1 -29235.814,E2 -29235.814} C_VEL
LIN {X 0,Y 55.147,Z 720.631,A -85,B 0,C 180,E1 -29242.666,E2 -29242.666} C_VEL
LIN {X 0,Y 52.408,Z 717.783,A -85,B 0,C 180,E1 -29253.832,E2 -29253.832} C_VEL
LIN {X 0,Y 51.774,Z 713.857,A -85,B 0,C 180,E1 -29265.739,E2 -29265.739} C_VEL
LIN {X 0,Y 53.495,Z 708.794,A -85,B 0,C 180,E1 -29277.361,E2 -29277.361} C_VEL
LIN {X 0,Y 57.384,Z 702.457,A -85,B 0,C 180,E1 -29287.745,E2 -29287.745} C_VEL
LIN {X 0,Y 62.978,Z 694.61,A -85,B 0,C 180,E1 -29296.483,E2 -29296.483} C_VEL
LIN {X 0,Y 68.597,Z 686.705,A -85,B 0,C 180,E1 -29302.408,E2 -29302.408} C_VEL
LIN {X 0,Y 75.122,Z 676.878,A -85,B 0,C 180,E1 -29307.334,E2 -29307.334} C_VEL
LIN {X 0,Y 81.31,Z 666.075,A -85,B 0,C 180,E1 -29311.044,E2 -29311.044} C_VEL
LIN {X 0,Y 86.333,Z 655.629,A -85,B 0,C 180,E1 -29313.55,E2 -29313.55} C_VEL
LIN {X 0,Y 91.106,Z 643.106,A -85,B 0,C 180,E1 -29315.656,E2 -29315.656} C_VEL
LIN {X 0,Y 94.821,Z 629.731,A -85,B 0,C 180,E1 -29317.22,E2 -29317.22} C_VEL
LIN {X 0,Y 96.639,Z 619.876,A -85,B 0,C 180,E1 -29318.072,E2 -29318.072} C_VEL
LIN {X 0,Y 97.95,Z 597.429,A -85,B 0,C 180,E1 -29320.472,E2 -29320.472} C_VEL
LIN {X 0,Y 98.585,Z 584.884,A -85,B 0,C 180,E1 -29321.765,E2 -29321.765} C_VEL
LIN {X 0,Y 98.483,Z 581.809,A -85,B 0,C 180,E1 -29322.405,E2 -29322.405} C_VEL
LIN {X 0,Y 97.742,Z 578.522,A -85,B 0,C 180,E1 -29323.93,E2 -29323.93} C_VEL
LIN {X 0,Y 96.765,Z 576.194,A -85,B 0,C 180,E1 -29325.729,E2 -29325.729} C_VEL
LIN {X 0,Y 95.684,Z 574.449,A -85,B 0,C 180,E1 -29327.754,E2 -29327.754} C_VEL
LIN {X 0,Y 91.834,Z 569.042,A -85,B 0,C 180,E1 -29337.913,E2 -29337.913} C_VEL
LIN {X 0,Y 91.219,Z 566.956,A -85,B 0,C 180,E1 -29341.653,E2 -29341.653} C_VEL
LIN {X 0,Y 90.668,Z 566.752,A -85,B 0,C 180,E1 -29348.917,E2 -29348.917} C_VEL
LIN {X 0,Y 91.165,Z 567.559,A -85,B 0,C 180,E1 -29354.75,E2 -29354.75} C_VEL
LIN {X 0,Y 92.709,Z 571.57,A -85,B 0,C 180,E1 -29361.978,E2 -29361.978} C_VEL
LIN {X 0,Y 94.407,Z 575.445,A -85,B 0,C 180,E1 -29366.723,E2 -29366.723} C_VEL
LIN {X 0,Y 96.37,Z 580.401,A -85,B 0,C 180,E1 -29370.97,E2 -29370.97} C_VEL
LIN {X 0,Y 97.393,Z 583.385,A -85,B 0,C 180,E1 -29372.918,E2 -29372.918} C_VEL
LIN {X 0,Y 95.036,Z 606.879,A -85,B 0,C 180,E1 -29374.396,E2 -29374.396} C_VEL
LIN {X 0,Y 92.432,Z 620.361,A -85,B 0,C 180,E1 -29375.733,E2 -29375.733} C_VEL
LIN {X 0,Y 88.71,Z 633.147,A -85,B 0,C 180,E1 -29377.618,E2 -29377.618} C_VEL
LIN {X 0,Y 83.783,Z 645.465,A -85,B 0,C 180,E1 -29380.067,E2 -29380.067} C_VEL
LIN {X 0,Y 78.331,Z 656.464,A -85,B 0,C 180,E1 -29383.212,E2 -29383.212} C_VEL
LIN {X 0,Y 72.343,Z 666.413,A -85,B 0,C 180,E1 -29387.166,E2 -29387.166} C_VEL
LIN {X 0,Y 66.061,Z 675.454,A -85,B 0,C 180,E1 -29392.299,E2 -29392.299} C_VEL
LIN {X 0,Y 59.199,Z 684.309,A -85,B 0,C 180,E1 -29399.712,E2 -29399.712} C_VEL
LIN {X 0,Y 53.353,Z 691.381,A -85,B 0,C 180,E1 -29408.669,E2 -29408.669} C_VEL
LIN {X 0,Y 49.445,Z 696.309,A -85,B 0,C 180,E1 -29417.704,E2 -29417.704} C_VEL
LIN {X 0,Y 46.396,Z 701.05,A -85,B 0,C 180,E1 -29430.015,E2 -29430.015} C_VEL
LIN {X 0,Y 45.501,Z 704.698,A -85,B 0,C 180,E1 -29443.412,E2 -29443.412} C_VEL
LIN {X 0,Y 46.933,Z 707.335,A -85,B 0,C 180,E1 -29456.711,E2 -29456.711} C_VEL
LIN {X 0,Y 51.33,Z 709.2,A -85,B 0,C 180,E1 -29470.586,E2 -29470.586} C_VEL
LIN {X 0,Y 50.364,Z 709.72,A -85,B 0,C 180,E1 -29474.263,E2 -29474.263} C_VEL
LIN {X 0,Y 44.742,Z 713.81,A -85,B 0,C 180,E1 -29510.966,E2 -29510.966} C_VEL
LIN {X 0,Y 48.826,Z 715.55,A -85,B 0,C 180,E1 -29528.8,E2 -29528.8} C_VEL
LIN {X 0,Y 52.831,Z 724.154,A -85,B 0,C 180,E1 -29540.547,E2 -29540.547} C_VEL
LIN {X 0,Y 59.882,Z 732.775,A -85,B 0,C 180,E1 -29551.883,E2 -29551.883} C_VEL
LIN {X 0,Y 65.275,Z 737.319,A -85,B 0,C 180,E1 -29557.309,E2 -29557.309} C_VEL
LIN {X 0,Y 63.778,Z 736.455,A -85,B 0,C 180,E1 -29559.507,E2 -29559.507} C_VEL
LIN {X 0,Y 56.196,Z 730.141,A -85,B 0,C 180,E1 -29571.28,E2 -29571.28} C_VEL
LIN {X 0,Y 51.796,Z 721.322,A -85,B 0,C 180,E1 -29588.6,E2 -29588.6} C_VEL
LIN {X 0,Y 50.568,Z 720.777,A -85,B 0,C 180,E1 -29593.848,E2 -29593.848} C_VEL
LIN {X 0,Y 47.979,Z 719.449,A -85,B 0,C 180,E1 -29601.563,E2 -29601.563} C_VEL
LIN {X 0,Y 45.183,Z 716.513,A -85,B 0,C 180,E1 -29614.446,E2 -29614.446} C_VEL
LIN {X 0,Y 45.097,Z 711.671,A -85,B 0,C 180,E1 -29630.755,E2 -29630.755} C_VEL
LIN {X 0,Y 48.491,Z 705.348,A -85,B 0,C 180,E1 -29645.415,E2 -29645.415} C_VEL
LIN {X 0,Y 53.846,Z 698.423,A -85,B 0,C 180,E1 -29655.86,E2 -29655.86} C_VEL
LIN {X 0,Y 60.708,Z 689.855,A -85,B 0,C 180,E1 -29664.113,E2 -29664.113} C_VEL
LIN {X 0,Y 67.289,Z 681.059,A -85,B 0,C 180,E1 -29669.484,E2 -29669.484} C_VEL
LIN {X 0,Y 74.395,Z 670.239,A -85,B 0,C 180,E1 -29673.803,E2 -29673.803} C_VEL
LIN {X 0,Y 80.336,Z 659.482,A -85,B 0,C 180,E1 -29676.696,E2 -29676.696} C_VEL
LIN {X 0,Y 85.693,Z 647.465,A -85,B 0,C 180,E1 -29678.869,E2 -29678.869} C_VEL
LIN {X 0,Y 89.902,Z 634.939,A -85,B 0,C 180,E1 -29680.486,E2 -29680.486} C_VEL
LIN {X 0,Y 92.952,Z 622.234,A -85,B 0,C 180,E1 -29681.577,E2 -29681.577} C_VEL
LIN {X 0,Y 94.29,Z 607.692,A -85,B 0,C 180,E1 -29683.215,E2 -29683.215} C_VEL
LIN {X 0,Y 95.639,Z 584.385,A -85,B 0,C 180,E1 -29685.756,E2 -29685.756} C_VEL
LIN {X 0,Y 94.25,Z 576.509,A -85,B 0,C 180,E1 -29689.769,E2 -29689.769} C_VEL
LIN {X 0,Y 93.482,Z 573.08,A -85,B 0,C 180,E1 -29692.166,E2 -29692.166} C_VEL
LIN {X 0,Y 92.193,Z 569.81,A -85,B 0,C 180,E1 -29696.447,E2 -29696.447} C_VEL
LIN {X 0,Y 91.834,Z 569.042,A -85,B 0,C 180,E1 -29697.913,E2 -29697.913} C_VEL
LIN {X 0,Y 91.342,Z 568.183,A -85,B 0,C 180,E1 -29700.27,E2 -29700.27} C_VEL
LIN {X 0,Y 90.887,Z 568.197,A -85,B 0,C 180,E1 -29702.717,E2 -29702.717} C_VEL
LIN {X 0,Y 90.371,Z 569.4,A -85,B 0,C 180,E1 -29706.4,E2 -29706.4} C_VEL
LIN {X 0,Y 90.647,Z 576.45,A -85,B 0,C 180,E1 -29717.457,E2 -29717.457} C_VEL
LIN {X 0,Y 91.417,Z 578.352,A -85,B 0,C 180,E1 -29720.821,E2 -29720.821} C_VEL
LIN {X 0,Y 92.777,Z 581.952,A -85,B 0,C 180,E1 -29725.204,E2 -29725.204} C_VEL
LIN {X 0,Y 94.289,Z 586.522,A -85,B 0,C 180,E1 -29729.045,E2 -29729.045} C_VEL
LIN {X 0,Y 94.141,Z 589.091,A -85,B 0,C 180,E1 -29729.358,E2 -29729.358} C_VEL
LIN {X 0,Y 91.91,Z 608.773,A -85,B 0,C 180,E1 -29730.54,E2 -29730.54} C_VEL
LIN {X 0,Y 89.301,Z 621.395,A -85,B 0,C 180,E1 -29731.751,E2 -29731.751} C_VEL
LIN {X 0,Y 85.895,Z 632.773,A -85,B 0,C 180,E1 -29733.315,E2 -29733.315} C_VEL
LIN {X 0,Y 80.912,Z 644.947,A -85,B 0,C 180,E1 -29735.496,E2 -29735.496} C_VEL
LIN {X 0,Y 75.122,Z 656.225,A -85,B 0,C 180,E1 -29738.431,E2 -29738.431} C_VEL
LIN {X 0,Y 68.749,Z 666.442,A -85,B 0,C 180,E1 -29742.186,E2 -29742.186} C_VEL
LIN {X 0,Y 61.943,Z 675.651,A -85,B 0,C 180,E1 -29747.113,E2 -29747.113} C_VEL
LIN {X 0,Y 54.377,Z 684.637,A -85,B 0,C 180,E1 -29754.452,E2 -29754.452} C_VEL
LIN {X 0,Y 47.713,Z 691.92,A -85,B 0,C 180,E1 -29763.791,E2 -29763.791} C_VEL
LIN {X 0,Y 42.47,Z 697.753,A -85,B 0,C 180,E1 -29775.644,E2 -29775.644} C_VEL
LIN {X 0,Y 39.219,Z 702.386,A -85,B 0,C 180,E1 -29790.017,E2 -29790.017} C_VEL
LIN {X 0,Y 38.538,Z 705.945,A -85,B 0,C 180,E1 -29805.894,E2 -29805.894} C_VEL
LIN {X 0,Y 40.605,Z 708.509,A -85,B 0,C 180,E1 -29821.301,E2 -29821.301} C_VEL
LIN {X 0,Y 43.376,Z 709.665,A -85,B 0,C 180,E1 -29830.418,E2 -29830.418} C_VEL
LIN {X 0,Y 41.239,Z 710.622,A -85,B 0,C 180,E1 -29837.029,E2 -29837.029} C_VEL
LIN {X 0,Y 38.844,Z 714.985,A -85,B 0,C 180,E1 -29880.004,E2 -29880.004} C_VEL
LIN {X 0,Y 45.294,Z 717.063,A -85,B 0,C 180,E1 -29899.383,E2 -29899.383} C_VEL
LIN {X 0,Y 54.437,Z 728.957,A -85,B 0,C 180,E1 -29915.522,E2 -29915.522} C_VEL
LIN {X 0,Y 56.88,Z 731.16,A -85,B 0,C 180,E1 -29918.158,E2 -29918.158} C_VEL
LIN {X 0,Y 49.997,Z 724.662,A -85,B 0,C 180,E1 -29930.744,E2 -29930.744} C_VEL
LIN {X 0,Y 47.347,Z 720.609,A -85,B 0,C 180,E1 -29939.304,E2 -29939.304} C_VEL
LIN {X 0,Y 43.787,Z 719.663,A -85,B 0,C 180,E1 -29951.26,E2 -29951.26} C_VEL
LIN {X 0,Y 40.838,Z 718.263,A -85,B 0,C 180,E1 -29960.074,E2 -29960.074} C_VEL
LIN {X 0,Y 37.979,Z 715.247,A -85,B 0,C 180,E1 -29975.291,E2 -29975.291} C_VEL
LIN {X 0,Y 38.239,Z 710.71,A -85,B 0,C 180,E1 -29993.215,E2 -29993.215} C_VEL
LIN {X 0,Y 41.956,Z 704.907,A -85,B 0,C 180,E1 -30008.894,E2 -30008.894} C_VEL
LIN {X 0,Y 47.945,Z 698.102,A -85,B 0,C 180,E1 -30020.293,E2 -30020.293} C_VEL
LIN {X 0,Y 55.452,Z 689.681,A -85,B 0,C 180,E1 -30028.791,E2 -30028.791} C_VEL
LIN {X 0,Y 62.489,Z 681.1,A -85,B 0,C 180,E1 -30034.099,E2 -30034.099} C_VEL
LIN {X 0,Y 69.99,Z 670.512,A -85,B 0,C 180,E1 -30038.226,E2 -30038.226} C_VEL
LIN {X 0,Y 76.992,Z 658.571,A -85,B 0,C 180,E1 -30041.243,E2 -30041.243} C_VEL
LIN {X 0,Y 82.573,Z 646.576,A -85,B 0,C 180,E1 -30043.208,E2 -30043.208} C_VEL
LIN {X 0,Y 86.973,Z 633.997,A -85,B 0,C 180,E1 -30044.684,E2 -30044.684} C_VEL
LIN {X 0,Y 90.078,Z 621.322,A -85,B 0,C 180,E1 -30045.756,E2 -30045.756} C_VEL
LIN {X 0,Y 91.629,Z 606.587,A -85,B 0,C 180,E1 -30047.401,E2 -30047.401} C_VEL
LIN {X 0,Y 92.996,Z 587.352,A -85,B 0,C 180,E1 -30049.457,E2 -30049.457} C_VEL
LIN {X 0,Y 92.036,Z 580.414,A -85,B 0,C 180,E1 -30053.283,E2 -30053.283} C_VEL
LIN {X 0,Y 91.665,Z 578.828,A -85,B 0,C 180,E1 -30054.705,E2 -30054.705} C_VEL
LIN {X 0,Y 90.794,Z 576.112,A -85,B 0,C 180,E1 -30058.433,E2 -30058.433} C_VEL
LIN {X 0,Y 90.211,Z 573.904,A -85,B 0,C 180,E1 -30062.469,E2 -30062.469} C_VEL
LIN {X 0,Y 89.884,Z 573.998,A -85,B 0,C 180,E1 -30071.195,E2 -30071.195} C_VEL
LIN {X 0,Y 90.163,Z 574.622,A -85,B 0,C 180,E1 -30074.079,E2 -30074.079} C_VEL
LIN {X 0,Y 90.647,Z 576.45,A -85,B 0,C 180,E1 -30077.457,E2 -30077.457} C_VEL
LIN {X 0,Y 91.075,Z 578.35,A -85,B 0,C 180,E1 -30079.763,E2 -30079.763} C_VEL
LIN {X 0,Y 91.498,Z 582.122,A -85,B 0,C 180,E1 -30082.307,E2 -30082.307} C_VEL
LIN {X 0,Y 91.683,Z 586.833,A -85,B 0,C 180,E1 -30084.203,E2 -30084.203} C_VEL
LIN {X 0,Y 91.517,Z 592.13,A -85,B 0,C 180,E1 -30085.337,E2 -30085.337} C_VEL
LIN {X 0,Y 91.404,Z 593.511,A -85,B 0,C 180,E1 -30085.474,E2 -30085.474} C_VEL
LIN {X 0,Y 89.236,Z 610.675,A -85,B 0,C 180,E1 -30086.452,E2 -30086.452} C_VEL
LIN {X 0,Y 86.319,Z 623.614,A -85,B 0,C 180,E1 -30087.635,E2 -30087.635} C_VEL
LIN {X 0,Y 82.395,Z 635.506,A -85,B 0,C 180,E1 -30089.203,E2 -30089.203} C_VEL
LIN {X 0,Y 77.051,Z 647.566,A -85,B 0,C 180,E1 -30091.245,E2 -30091.245} C_VEL
LIN {X 0,Y 70.971,Z 658.533,A -85,B 0,C 180,E1 -30093.986,E2 -30093.986} C_VEL
LIN {X 0,Y 64.224,Z 668.452,A -85,B 0,C 180,E1 -30097.517,E2 -30097.517} C_VEL
LIN {X 0,Y 56.96,Z 677.487,A -85,B 0,C 180,E1 -30102.261,E2 -30102.261} C_VEL
LIN {X 0,Y 48.771,Z 686.338,A -85,B 0,C 180,E1 -30109.593,E2 -30109.593} C_VEL
LIN {X 0,Y 41.456,Z 693.45,A -85,B 0,C 180,E1 -30119.449,E2 -30119.449} C_VEL
LIN {X 0,Y 35.588,Z 699.174,A -85,B 0,C 180,E1 -30132.789,E2 -30132.789} C_VEL
LIN {X 0,Y 32.026,Z 703.718,A -85,B 0,C 180,E1 -30150.021,E2 -30150.021} C_VEL
LIN {X 0,Y 31.383,Z 706.151,A -85,B 0,C 180,E1 -30162.963,E2 -30162.963} C_VEL
LIN {X 0,Y 33.527,Z 709.105,A -85,B 0,C 180,E1 -30183.027,E2 -30183.027} C_VEL
LIN {X 0,Y 34.623,Z 709.669,A -85,B 0,C 180,E1 -30187.538,E2 -30187.538} C_VEL
LIN {X 0,Y 34.092,Z 710.585,A -85,B 0,C 180,E1 -30194.616,E2 -30194.616} C_VEL
LIN {X 0,Y 31.45,Z 714.888,A -85,B 0,C 180,E1 -30240.005,E2 -30240.005} C_VEL
LIN {X 0,Y 43.669,Z 718.396,A -85,B 0,C 180,E1 -30271.541,E2 -30271.541} C_VEL
LIN {X 0,Y 48.375,Z 723.666,A -85,B 0,C 180,E1 -30278.553,E2 -30278.553} C_VEL
LIN {X 0,Y 47.351,Z 722.748,A -85,B 0,C 180,E1 -30282.067,E2 -30282.067} C_VEL
LIN {X 0,Y 44.422,Z 719.744,A -85,B 0,C 180,E1 -30288.489,E2 -30288.489} C_VEL
LIN {X 0,Y 39.937,Z 719.301,A -85,B 0,C 180,E1 -30298.115,E2 -30298.115} C_VEL
LIN {X 0,Y 37.108,Z 718.528,A -85,B 0,C 180,E1 -30307.722,E2 -30307.722} C_VEL
LIN {X 0,Y 33.731,Z 717.077,A -85,B 0,C 180,E1 -30317.954,E2 -30317.954} C_VEL
LIN {X 0,Y 30.752,Z 713.974,A -85,B 0,C 180,E1 -30336.539,E2 -30336.539} C_VEL
LIN {X 0,Y 31.499,Z 709.733,A -85,B 0,C 180,E1 -30356.804,E2 -30356.804} C_VEL
LIN {X 0,Y 36.634,Z 703.42,A -85,B 0,C 180,E1 -30375.979,E2 -30375.979} C_VEL
LIN {X 0,Y 43.707,Z 696.512,A -85,B 0,C 180,E1 -30387.556,E2 -30387.556} C_VEL
LIN {X 0,Y 52.083,Z 687.959,A -85,B 0,C 180,E1 -30395.589,E2 -30395.589} C_VEL
LIN {X 0,Y 59.718,Z 679.196,A -85,B 0,C 180,E1 -30400.269,E2 -30400.269} C_VEL
LIN {X 0,Y 67.657,Z 668.378,A -85,B 0,C 180,E1 -30403.88,E2 -30403.88} C_VEL
LIN {X 0,Y 74.175,Z 657.641,A -85,B 0,C 180,E1 -30406.169,E2 -30406.169} C_VEL
LIN {X 0,Y 79.964,Z 645.656,A -85,B 0,C 180,E1 -30407.854,E2 -30407.854} C_VEL
LIN {X 0,Y 84.518,Z 633.072,A -85,B 0,C 180,E1 -30409.144,E2 -30409.144} C_VEL
LIN {X 0,Y 87.49,Z 621.541,A -85,B 0,C 180,E1 -30410.01,E2 -30410.01} C_VEL
LIN {X 0,Y 89.231,Z 608.156,A -85,B 0,C 180,E1 -30411.52,E2 -30411.52} C_VEL
LIN {X 0,Y 90.69,Z 590.033,A -85,B 0,C 180,E1 -30413.539,E2 -30413.539} C_VEL
LIN {X 0,Y 90.237,Z 585.215,A -85,B 0,C 180,E1 -30416.436,E2 -30416.436} C_VEL
LIN {X 0,Y 89.534,Z 582.548,A -85,B 0,C 180,E1 -30420.28,E2 -30420.28} C_VEL
LIN {X 0,Y 89.17,Z 580.892,A -85,B 0,C 180,E1 -30423.67,E2 -30423.67} C_VEL
LIN {X 0,Y 89.012,Z 581.062,A -85,B 0,C 180,E1 -30431.306,E2 -30431.306} C_VEL
LIN {X 0,Y 89.147,Z 581.548,A -85,B 0,C 180,E1 -30433.079,E2 -30433.079} C_VEL
LIN {X 0,Y 90.069,Z 584.876,A -85,B 0,C 180,E1 -30439.215,E2 -30439.215} C_VEL
LIN {X 0,Y 91.166,Z 588.296,A -85,B 0,C 180,E1 -30443.469,E2 -30443.469} C_VEL
LIN {X 0,Y 91.712,Z 590.26,A -85,B 0,C 180,E1 -30445.238,E2 -30445.238} C_VEL
LIN {X 0,Y 91.404,Z 593.511,A -85,B 0,C 180,E1 -30445.474,E2 -30445.474} C_VEL
LIN {X 0,Y 90.937,Z 597.415,A -85,B 0,C 180,E1 -30445.542,E2 -30445.542} C_VEL
LIN {X 0,Y 89.487,Z 605.103,A -85,B 0,C 180,E1 -30444.767,E2 -30444.767} C_VEL
LIN {X 0,Y 85.974,Z 618.294,A -85,B 0,C 180,E1 -30443.005,E2 -30443.005} C_VEL
LIN {X 0,Y 84.33,Z 623.957,A -85,B 0,C 180,E1 -30443.084,E2 -30443.084} C_VEL
LIN {X 0,Y 80.111,Z 636.351,A -85,B 0,C 180,E1 -30444.491,E2 -30444.491} C_VEL
LIN {X 0,Y 74.457,Z 648.617,A -85,B 0,C 180,E1 -30446.294,E2 -30446.294} C_VEL
LIN {X 0,Y 68.077,Z 659.575,A -85,B 0,C 180,E1 -30448.678,E2 -30448.678} C_VEL
LIN {X 0,Y 60.175,Z 670.459,A -85,B 0,C 180,E1 -30452.162,E2 -30452.162} C_VEL
LIN {X 0,Y 52.486,Z 679.314,A -85,B 0,C 180,E1 -30456.564,E2 -30456.564} C_VEL
LIN {X 0,Y 43.608,Z 688.002,A -85,B 0,C 180,E1 -30463.534,E2 -30463.534} C_VEL
LIN {X 0,Y 35.517,Z 694.969,A -85,B 0,C 180,E1 -30473.609,E2 -30473.609} C_VEL
LIN {X 0,Y 28.835,Z 700.597,A -85,B 0,C 180,E1 -30488.581,E2 -30488.581} C_VEL
LIN {X 0,Y 24.842,Z 705.051,A -85,B 0,C 180,E1 -30510.027,E2 -30510.027} C_VEL
LIN {X 0,Y 24.413,Z 707.441,A -85,B 0,C 180,E1 -30526.76,E2 -30526.76} C_VEL
LIN {X 0,Y 27.259,Z 710.088,A -85,B 0,C 180,E1 -30549.341,E2 -30549.341} C_VEL
LIN {X 0,Y 23.053,Z 713.059,A -85,B 0,C 180,E1 -30582.257,E2 -30582.257} C_VEL
LIN {X 0,Y 31.14,Z 716.783,A -85,B 0,C 180,E1 -30626.837,E2 -30626.837} C_VEL
LIN {X 0,Y 39.045,Z 718.456,A -85,B 0,C 180,E1 -30639.055,E2 -30639.055} C_VEL
LIN {X 0,Y 38.47,Z 718.61,A -85,B 0,C 180,E1 -30643.025,E2 -30643.025} C_VEL
LIN {X 0,Y 34.167,Z 718.213,A -85,B 0,C 180,E1 -30651.872,E2 -30651.872} C_VEL
LIN {X 0,Y 30.611,Z 717.389,A -85,B 0,C 180,E1 -30662.641,E2 -30662.641} C_VEL
LIN {X 0,Y 25.204,Z 714.915,A -85,B 0,C 180,E1 -30681.959,E2 -30681.959} C_VEL
LIN {X 0,Y 23.553,Z 711.37,A -85,B 0,C 180,E1 -30707.331,E2 -30707.331} C_VEL
LIN {X 0,Y 26.708,Z 706.726,A -85,B 0,C 180,E1 -30731.102,E2 -30731.102} C_VEL
LIN {X 0,Y 33.346,Z 700.874,A -85,B 0,C 180,E1 -30747.424,E2 -30747.424} C_VEL
LIN {X 0,Y 41.785,Z 693.564,A -85,B 0,C 180,E1 -30757.636,E2 -30757.636} C_VEL
LIN {X 0,Y 51.144,Z 684.477,A -85,B 0,C 180,E1 -30764.084,E2 -30764.084} C_VEL
LIN {X 0,Y 59.353,Z 675.229,A -85,B 0,C 180,E1 -30767.602,E2 -30767.602} C_VEL
LIN {X 0,Y 66.877,Z 664.947,A -85,B 0,C 180,E1 -30770.072,E2 -30770.072} C_VEL
LIN {X 0,Y 73.651,Z 653.51,A -85,B 0,C 180,E1 -30771.83,E2 -30771.83} C_VEL
LIN {X 0,Y 78.742,Z 642.7,A -85,B 0,C 180,E1 -30772.965,E2 -30772.965} C_VEL
LIN {X 0,Y 83.23,Z 630.084,A -85,B 0,C 180,E1 -30773.997,E2 -30773.997} C_VEL
LIN {X 0,Y 85.517,Z 621.123,A -85,B 0,C 180,E1 -30774.573,E2 -30774.573} C_VEL
LIN {X 0,Y 87.535,Z 607.157,A -85,B 0,C 180,E1 -30776.156,E2 -30776.156} C_VEL
LIN {X 0,Y 88.873,Z 593.157,A -85,B 0,C 180,E1 -30777.591,E2 -30777.591} C_VEL
LIN {X 0,Y 88.724,Z 590.78,A -85,B 0,C 180,E1 -30779.289,E2 -30779.289} C_VEL
LIN {X 0,Y 88.283,Z 588.382,A -85,B 0,C 180,E1 -30783.279,E2 -30783.279} C_VEL
LIN {X 0,Y 88.201,Z 587.866,A -85,B 0,C 180,E1 -30784.569,E2 -30784.569} C_VEL
